FUNCTION "FC13 - MANUAL" : VOID	// FC 13
TITLE = Manual commands
VERSION : 0.1
BEGIN
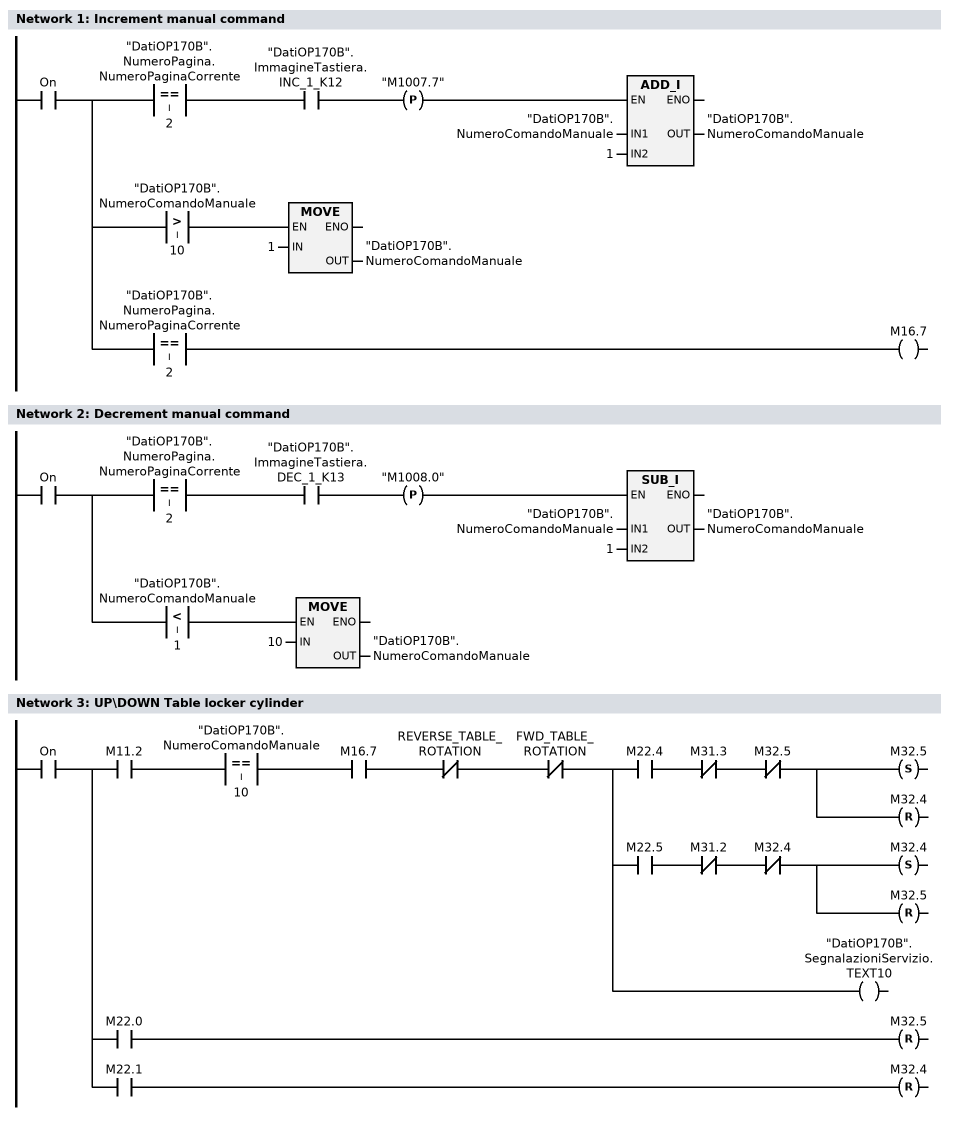
NETWORK
TITLE = Increment manual command
      A     "On";
      =     L 1.0;
      A     L 1.0;
      A(;
      L     "DatiOP170B".NumeroPagina.NumeroPaginaCorrente;
      L     2;
      ==I;
      );
      A     "DatiOP170B".ImmagineTastiera.INC_1_K12;
      FP    "M1007.7";
      JNB   _001;
      L     "DatiOP170B".NumeroComandoManuale;
      L     1;
      +I;
      T     "DatiOP170B".NumeroComandoManuale;
_001: NOP   0;
      A     L 1.0;
      A(;
      L     "DatiOP170B".NumeroComandoManuale;
      L     10;
      >I;
      );
      JNB   _002;
      L     1;
      T     "DatiOP170B".NumeroComandoManuale;
_002: NOP   0;
      A     L 1.0;
      A(;
      L     "DatiOP170B".NumeroPagina.NumeroPaginaCorrente;
      L     2;
      ==I;
      );
      =     "M16.7";
NETWORK
TITLE = Decrement manual command
      A     "On";
      =     L 1.0;
      A     L 1.0;
      A(;
      L     "DatiOP170B".NumeroPagina.NumeroPaginaCorrente;
      L     2;
      ==I;
      );
      A     "DatiOP170B".ImmagineTastiera.DEC_1_K13;
      FP    "M1008.0";
      JNB   _003;
      L     "DatiOP170B".NumeroComandoManuale;
      L     1;
      -I;
      T     "DatiOP170B".NumeroComandoManuale;
_003: NOP   0;
      A     L 1.0;
      A(;
      L     "DatiOP170B".NumeroComandoManuale;
      L     1;
      <I;
      );
      JNB   _004;
      L     10;
      T     "DatiOP170B".NumeroComandoManuale;
_004: NOP   0;
NETWORK
TITLE = UP\DOWN Table locker cylinder
      A     "On";
      =     L 1.0;
      A     L 1.0;
      A     "M11.2";
      A(;
      L     "DatiOP170B".NumeroComandoManuale;
      L     10;
      ==I;
      );
      A     "M16.7";
      AN    "REVERSE_TABLE_ROTATION";
      AN    "FWD_TABLE_ROTATION";
      =     L 1.1;
      A     L 1.1;
      A     "M22.4";
      AN    "M31.3";
      AN    "M32.5";
      S     "M32.5";
      R     "M32.4";
      A     L 1.1;
      A     "M22.5";
      AN    "M31.2";
      AN    "M32.4";
      S     "M32.4";
      R     "M32.5";
      A     L 1.1;
      BLD   102;
      =     "DatiOP170B".SegnalazioniServizio.TEXT10;
      A     L 1.0;
      A     "M22.0";
      R     "M32.5";
      A     L 1.0;
      A     "M22.1";
      R     "M32.4";
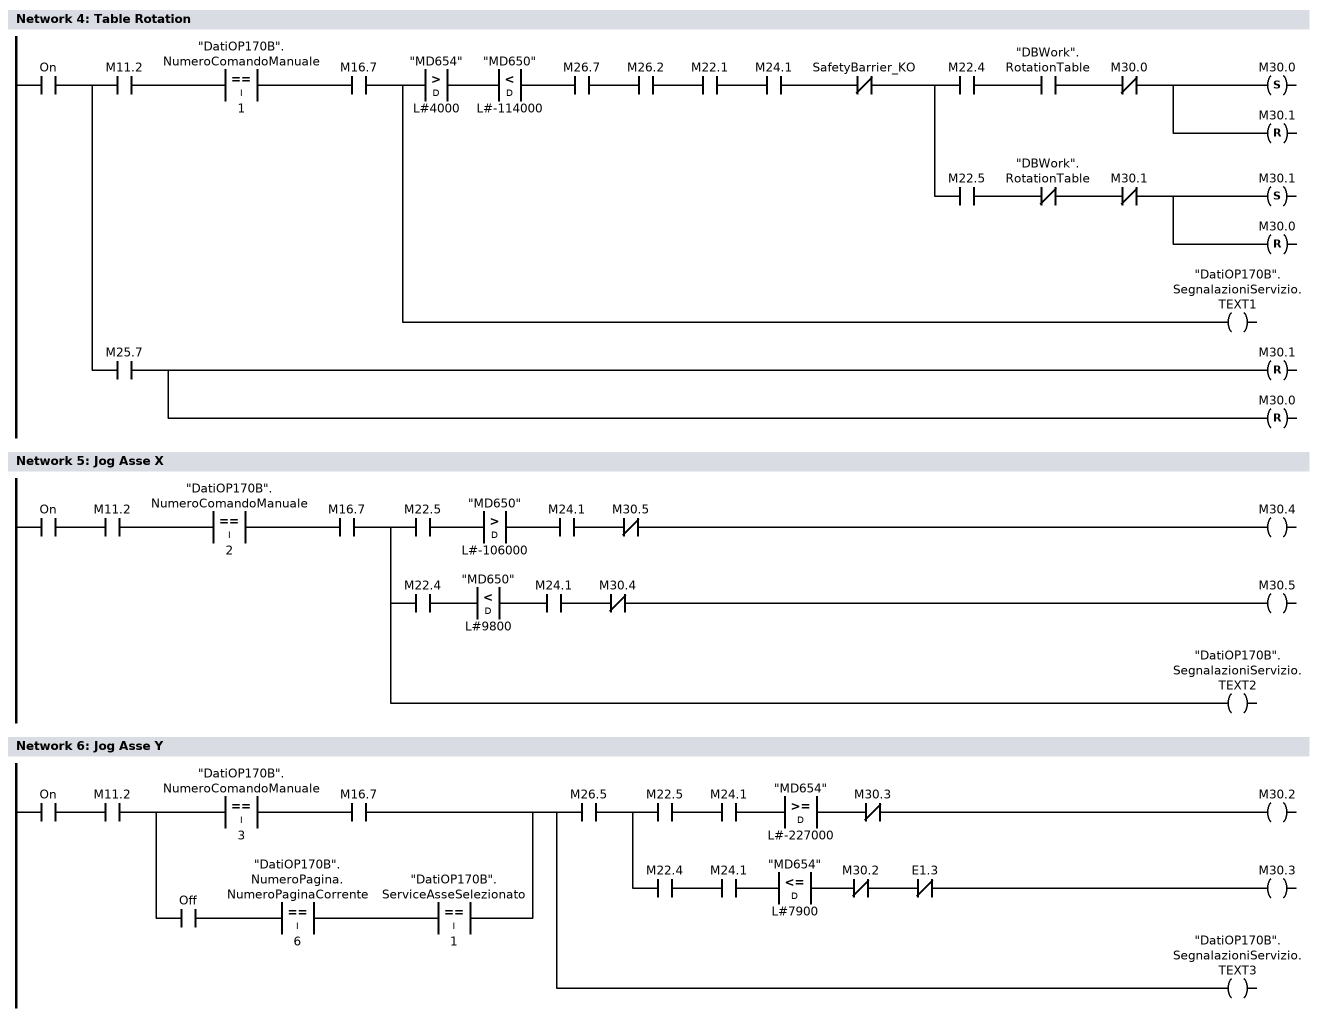
NETWORK
TITLE = Table Rotation
      A     "On";
      =     L 1.0;
      A     L 1.0;
      A     "M11.2";
      A(;
      L     "DatiOP170B".NumeroComandoManuale;
      L     1;
      ==I;
      );
      A     "M16.7";
      =     L 1.1;
      A     L 1.1;
      A(;
      L     "MD654";
      L     L#4000;
      >D;
      );
      A(;
      L     "MD650";
      L     L#-114000;
      <D;
      );
      A     "M26.7";
      A     "M26.2";
      A     "M22.1";
      A     "M24.1";
      AN    "SafetyBarrier_KO";
      =     L 1.2;
      A     L 1.2;
      A     "M22.4";
      A     "DBWork".RotationTable;
      AN    "M30.0";
      S     "M30.0";
      R     "M30.1";
      A     L 1.2;
      A     "M22.5";
      AN    "DBWork".RotationTable;
      AN    "M30.1";
      S     "M30.1";
      R     "M30.0";
      A     L 1.1;
      BLD   102;
      =     "DatiOP170B".SegnalazioniServizio.TEXT1;
      A     L 1.0;
      A     "M25.7";
      R     "M30.1";
      R     "M30.0";
NETWORK
TITLE = Jog Asse X
      A     "On";
      A     "M11.2";
      A(;
      A(;
      L     "DatiOP170B".NumeroComandoManuale;
      L     2;
      ==I;
      );
      A     "M16.7";
      );
      =     L 0.0;
      A     L 0.0;
      A     "M22.5";
      A(;
      L     "MD650";
      L     L#-106000;
      >D;
      );
      A     "M24.1";
      AN    "M30.5";
      =     "M30.4";
      A     L 0.0;
      A     "M22.4";
      A(;
      L     "MD650";
      L     L#9800;
      <D;
      );
      A     "M24.1";
      AN    "M30.4";
      =     "M30.5";
      A     L 0.0;
      BLD   102;
      =     "DatiOP170B".SegnalazioniServizio.TEXT2;
NETWORK
TITLE = Jog Asse Y
      A     "On";
      A     "M11.2";
      A(;
      A(;
      L     "DatiOP170B".NumeroComandoManuale;
      L     3;
      ==I;
      );
      A     "M16.7";
      O;
      A     "Off";
      A(;
      L     "DatiOP170B".NumeroPagina.NumeroPaginaCorrente;
      L     6;
      ==I;
      );
      A(;
      L     "DatiOP170B".ServiceAsseSelezionato;
      L     1;
      ==I;
      );
      );
      =     L 0.0;
      A     L 0.0;
      A     "M26.5";
      =     L 0.1;
      A     L 0.1;
      A     "M22.5";
      A     "M24.1";
      A(;
      L     "MD654";
      L     L#-227000;
      >=D;
      );
      AN    "M30.3";
      =     "M30.2";
      A     L 0.1;
      A     "M22.4";
      A     "M24.1";
      A(;
      L     "MD654";
      L     L#7900;
      <=D;
      );
      AN    "M30.2";
      AN    "E1.3";
      =     "M30.3";
      A     L 0.0;
      BLD   102;
      =     "DatiOP170B".SegnalazioniServizio.TEXT3;
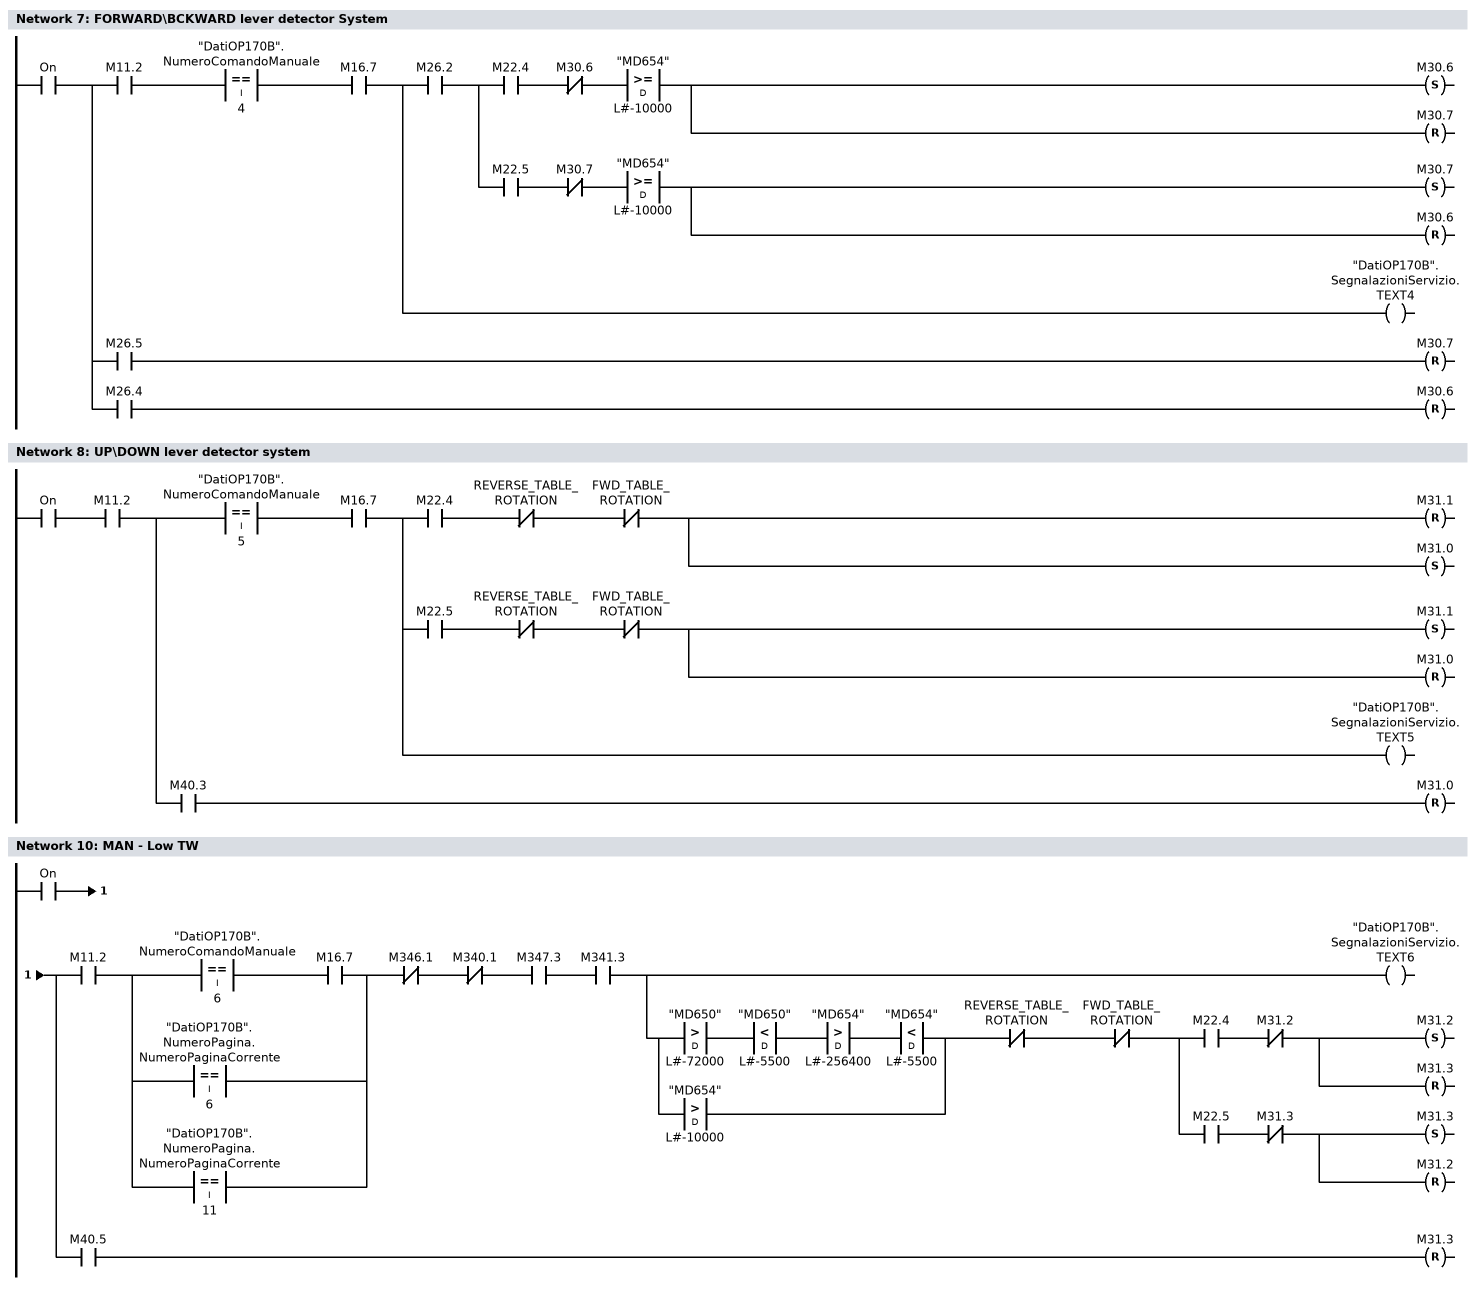
NETWORK
TITLE = FORWARD\BCKWARD lever detector System
//controllo fuori ingombro asse Y
      A     "On";
      =     L 1.0;
      A     L 1.0;
      A     "M11.2";
      A(;
      L     "DatiOP170B".NumeroComandoManuale;
      L     4;
      ==I;
      );
      A     "M16.7";
      =     L 1.1;
      A     L 1.1;
      A     "M26.2";
      =     L 1.2;
      A     L 1.2;
      A     "M22.4";
      AN    "M30.6";
      A(;
      L     "MD654";
      L     L#-10000;
      >=D;
      );
      S     "M30.6";
      R     "M30.7";
      A     L 1.2;
      A     "M22.5";
      AN    "M30.7";
      A(;
      L     "MD654";
      L     L#-10000;
      >=D;
      );
      S     "M30.7";
      R     "M30.6";
      A     L 1.1;
      BLD   102;
      =     "DatiOP170B".SegnalazioniServizio.TEXT4;
      A     L 1.0;
      A     "M26.5";
      R     "M30.7";
      A     L 1.0;
      A     "M26.4";
      R     "M30.6";
NETWORK
TITLE = UP\DOWN lever detector system
      A     "On";
      A     "M11.2";
      =     L 1.0;
      A     L 1.0;
      A(;
      L     "DatiOP170B".NumeroComandoManuale;
      L     5;
      ==I;
      );
      A     "M16.7";
      =     L 1.1;
      A     L 1.1;
      A     "M22.4";
      AN    "REVERSE_TABLE_ROTATION";
      AN    "FWD_TABLE_ROTATION";
      R     "M31.1";
      S     "M31.0";
      A     L 1.1;
      A     "M22.5";
      AN    "REVERSE_TABLE_ROTATION";
      AN    "FWD_TABLE_ROTATION";
      S     "M31.1";
      R     "M31.0";
      A     L 1.1;
      BLD   102;
      =     "DatiOP170B".SegnalazioniServizio.TEXT5;
      A     L 1.0;
      A     "M40.3";
      R     "M31.0";
NETWORK
TITLE = UP\DOWN Torch Welding Machine
//      U     "On"
//      =     L      0.0
//      U     L      0.0
//      U     "M11.2"
//      U(    
//      U(    
//      L     "DatiOP170B".NumeroComandoManuale
//      L     6
//      ==I   
//      )     
//      U     "M16.7"
//      O     
//      U(    
//      O(    
//      L     "DatiOP170B".NumeroPagina.NumeroPaginaCorrente
//      L     6
//      ==I   
//      )     
//      O(    
//      L     "DatiOP170B".NumeroPagina.NumeroPaginaCorrente
//      L     11
//      ==I   
//      )     
//      )     
//      UN    "M346.1"
//      UN    "M340.1"
//      U     "M347.3"
//      U     "M341.3"
//      )     
//      =     L      0.1
//      U     L      0.1
//      U(    
//      U(    
//      L     "MD650"
//      L     L#-72000
//      >D    
//      )     
//      U(    
//      L     "MD650"
//      L     L#-5500
//      <D    
//      )     
//      U(    
//      L     "MD654"
//      L     L#-256400
//      >D    
//      )     
//      U(    
//      L     "MD654"
//      L     L#-5500
//      <D    
//      )     
//      O(    
//      L     "MD654"
//      L     -10000
//      >D    
//      )     
//      )     
//      UN    "REVERSE_TABLE_ROTATION"
//      UN    "FWD_TABLE_ROTATION"
//      =     L      0.2
//      U     L      0.2
//      U     "M22.4"
//      UN    "M31.2"
//      S     "M31.2"
//      R     "M31.3"
//      U     L      0.2
//      U     "M22.5"
//      UN    "M31.3"
//      S     "M31.3"
//      R     "M31.2"
//      U     L      0.1
//      BLD   102
//      =     "DatiOP170B".SegnalazioniServizio.TEXT6
//      U     L      0.0
//      U     "M40.5"
//      R     "M31.3"
//  A     L      0.0
// A     "M24.1"
// R     "M31.2"
NETWORK
TITLE = MAN - Low TW
      A     "On";
      =     L 1.0;
      A     L 1.0;
      A     "M11.2";
      A(;
      A(;
      L     "DatiOP170B".NumeroComandoManuale;
      L     6;
      ==I;
      );
      A     "M16.7";
      O(;
      L     "DatiOP170B".NumeroPagina.NumeroPaginaCorrente;
      L     6;
      ==I;
      );
      O(;
      L     "DatiOP170B".NumeroPagina.NumeroPaginaCorrente;
      L     11;
      ==I;
      );
      );
      AN    "M346.1";
      AN    "M340.1";
      A     "M347.3";
      A     "M341.3";
      =     L 1.1;
      A     L 1.1;
      BLD   102;
      =     "DatiOP170B".SegnalazioniServizio.TEXT6;
      A     L 1.1;
      A(;
      A(;
      L     "MD650";
      L     L#-72000;
      >D;
      );
      A(;
      L     "MD650";
      L     L#-5500;
      <D;
      );
      A(;
      L     "MD654";
      L     L#-256400;
      >D;
      );
      A(;
      L     "MD654";
      L     L#-5500;
      <D;
      );
      O(;
      L     "MD654";
      L     L#-10000;
      >D;
      );
      );
      AN    "REVERSE_TABLE_ROTATION";
      AN    "FWD_TABLE_ROTATION";
      =     L 1.2;
      A     L 1.2;
      A     "M22.4";
      AN    "M31.2";
      S     "M31.2";
      R     "M31.3";
      A     L 1.2;
      A     "M22.5";
      AN    "M31.3";
      S     "M31.3";
      R     "M31.2";
      A     L 1.0;
      A     "M40.5";
      R     "M31.3";
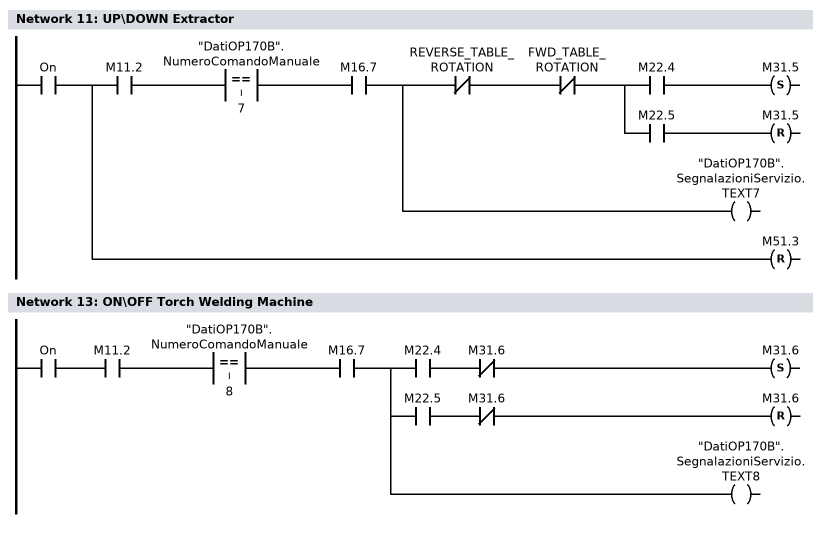
NETWORK
TITLE = UP\DOWN Extractor
      A     "On";
      =     L 1.0;
      A     L 1.0;
      A     "M11.2";
      A(;
      L     "DatiOP170B".NumeroComandoManuale;
      L     7;
      ==I;
      );
      A     "M16.7";
      =     L 1.1;
      A     L 1.1;
      AN    "REVERSE_TABLE_ROTATION";
      AN    "FWD_TABLE_ROTATION";
      =     L 1.2;
      A     L 1.2;
      A     "M22.4";
      S     "M31.5";
      A     L 1.2;
      A     "M22.5";
      R     "M31.5";
      A     L 1.1;
      BLD   102;
      =     "DatiOP170B".SegnalazioniServizio.TEXT7;
      A     L 1.0;
      BLD   102;
      R     "M51.3";
NETWORK
TITLE =
NETWORK
TITLE = ON\OFF Torch Welding Machine
      A     "On";
      A     "M11.2";
      A(;
      L     "DatiOP170B".NumeroComandoManuale;
      L     8;
      ==I;
      );
      A     "M16.7";
      =     L 1.0;
      A     L 1.0;
      A     "M22.4";
      AN    "M31.6";
      S     "M31.6";
      A     L 1.0;
      A     "M22.5";
      AN    "M31.6";
      R     "M31.6";
      A     L 1.0;
      BLD   102;
      =     "DatiOP170B".SegnalazioniServizio.TEXT8;
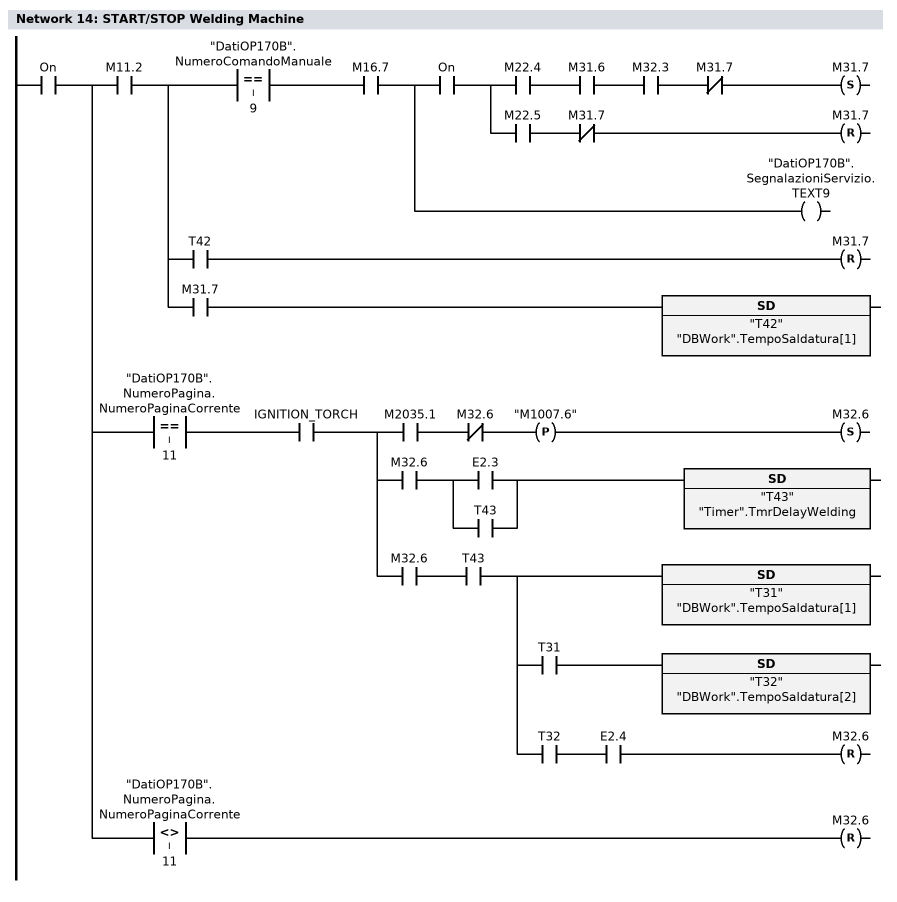
NETWORK
TITLE = START/STOP Welding Machine
      A     "On";
      =     L 1.0;
      A     L 1.0;
      A     "M11.2";
      =     L 1.1;
      A     L 1.1;
      A(;
      L     "DatiOP170B".NumeroComandoManuale;
      L     9;
      ==I;
      );
      A     "M16.7";
      =     L 1.2;
      A     L 1.2;
      A     "On";
      =     L 1.3;
      A     L 1.3;
      A     "M22.4";
      A     "M31.6";
      A     "M32.3";
      AN    "M31.7";
      S     "M31.7";
      A     L 1.3;
      A     "M22.5";
      AN    "M31.7";
      R     "M31.7";
      A     L 1.2;
      BLD   102;
      =     "DatiOP170B".SegnalazioniServizio.TEXT9;
      A     L 1.1;
      A     "T42";
      R     "M31.7";
      A     L 1.1;
      A     "M31.7";
      L     "DBWork".TempoSaldatura[1];
      SD    "T42";
      A     L 1.0;
      A(;
      L     "DatiOP170B".NumeroPagina.NumeroPaginaCorrente;
      L     11;
      ==I;
      );
      A     "IGNITION_TORCH";
      =     L 1.1;
      A     L 1.1;
      A     "M2035.1";
      AN    "M32.6";
      FP    "M1007.6";
      S     "M32.6";
      A     L 1.1;
      A     "M32.6";
      A(;
      O     "E2.3";
      O     "T43";
      );
      L     "Timer".TmrDelayWelding;
      SD    "T43";
      A     L 1.1;
      A     "M32.6";
      A     "T43";
      =     L 1.2;
      A     L 1.2;
      BLD   102;
      L     "DBWork".TempoSaldatura[1];
      SD    "T31";
      A     L 1.2;
      A     "T31";
      L     "DBWork".TempoSaldatura[2];
      SD    "T32";
      A     L 1.2;
      A     "T32";
      A     "E2.4";
      R     "M32.6";
      A     L 1.0;
      A(;
      L     "DatiOP170B".NumeroPagina.NumeroPaginaCorrente;
      L     11;
      <>I;
      );
      R     "M32.6";
END_FUNCTION

FUNCTION "FC14 - AUTOMATIC" : VOID	// FC 14
TITLE = Automatic cycle management
VERSION : 0.1
VAR_TEMP
  MinX : DINT ;
  MinY : DINT ;
  MaxX : DINT ;
  MaxY : DINT ;
END_VAR
BEGIN
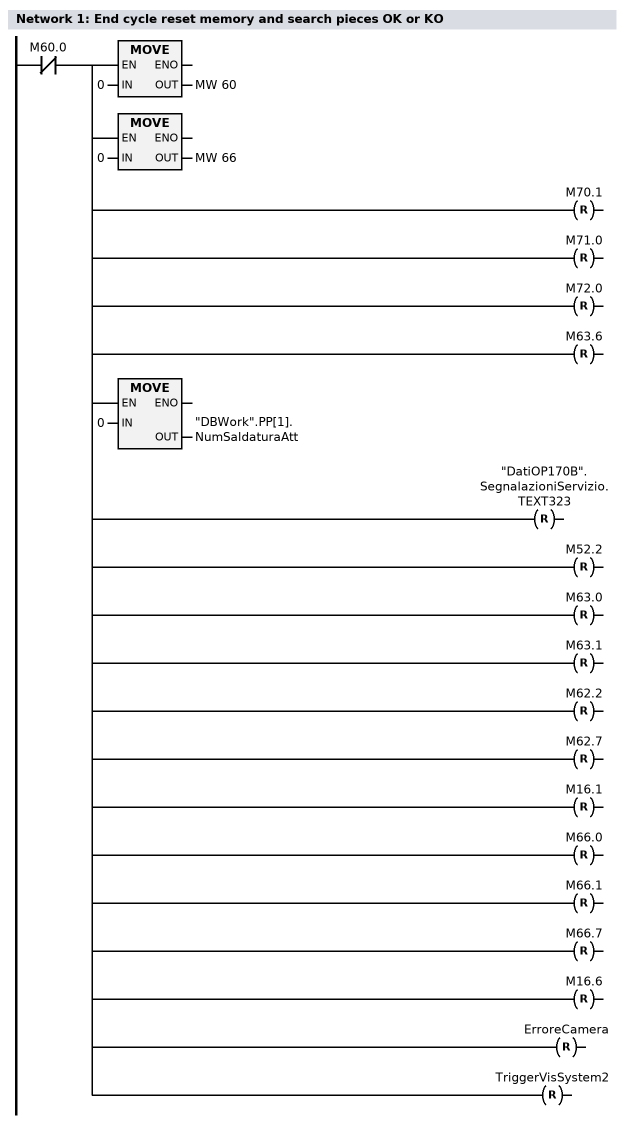
NETWORK
TITLE = End cycle reset memory and search pieces OK or KO
      AN    "M60.0";
      =     L 16.0;
      A     L 16.0;
      JNB   _001;
      L     0;
      T     MW 60;
_001: NOP   0;
      A     L 16.0;
      JNB   _002;
      L     0;
      T     MW 66;
_002: NOP   0;
      A     L 16.0;
      BLD   102;
      R     "M70.1";
      A     L 16.0;
      BLD   102;
      R     "M71.0";
      A     L 16.0;
      BLD   102;
      R     "M72.0";
      A     L 16.0;
      BLD   102;
      R     "M63.6";
      A     L 16.0;
      JNB   _003;
      L     0;
      T     "DBWork".PP[1].NumSaldaturaAtt;
_003: NOP   0;
      A     L 16.0;
      BLD   102;
      R     "DatiOP170B".SegnalazioniServizio.TEXT323;
      A     L 16.0;
      BLD   102;
      R     "M52.2";
      A     L 16.0;
      BLD   102;
      R     "M63.0";
      A     L 16.0;
      BLD   102;
      R     "M63.1";
      A     L 16.0;
      BLD   102;
      R     "M62.2";
      A     L 16.0;
      BLD   102;
      R     "M62.7";
      A     L 16.0;
      BLD   102;
      R     "M16.1";
      A     L 16.0;
      BLD   102;
      R     "M66.0";
      A     L 16.0;
      BLD   102;
      R     "M66.1";
      A     L 16.0;
      BLD   102;
      R     "M66.7";
      A     L 16.0;
      BLD   102;
      R     "M16.6";
      A     L 16.0;
      BLD   102;
      R     "ErroreCamera";
      A     L 16.0;
      BLD   102;
      R     "TriggerVisSystem2";
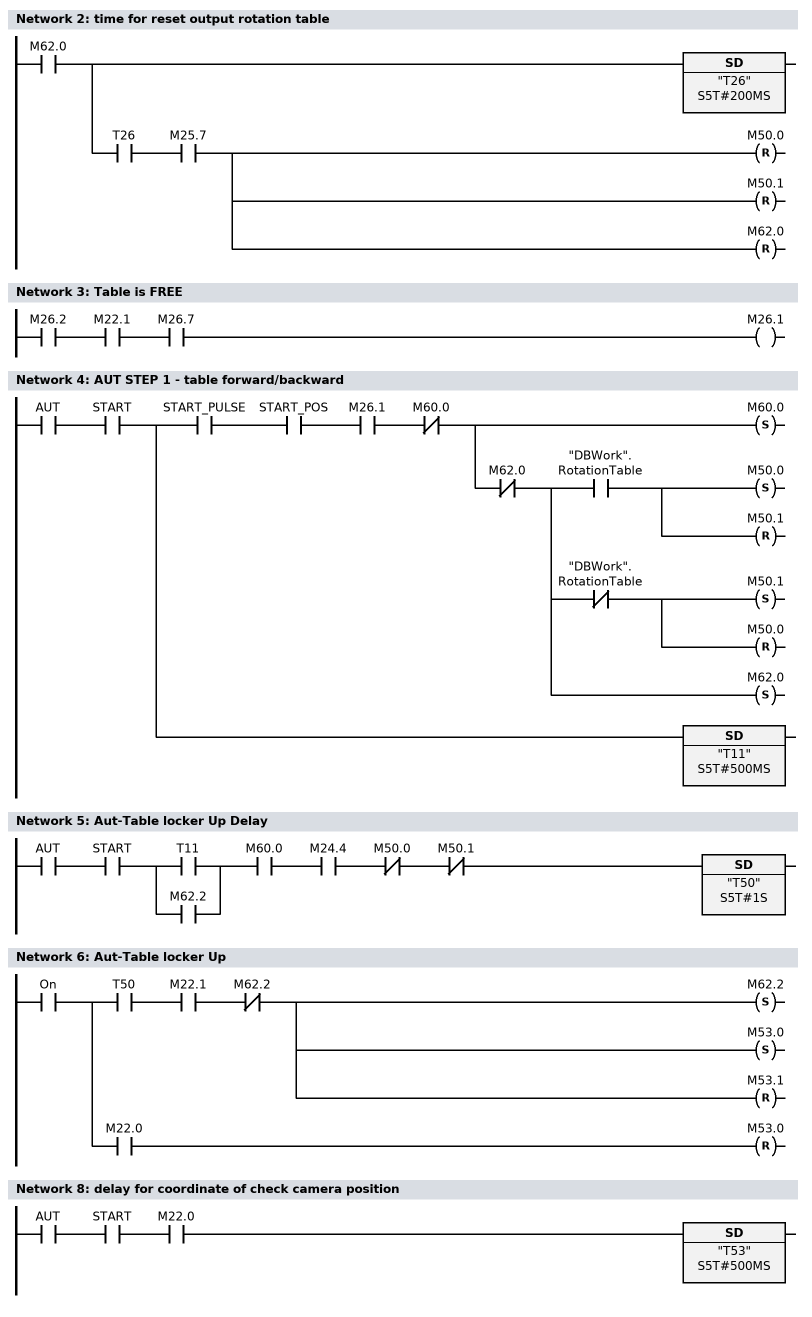
NETWORK
TITLE = time for reset output rotation table
//Reset Output Rotation Table 
      A     "M62.0";
      =     L 16.0;
      A     L 16.0;
      BLD   102;
      L     S5T#200MS;
      SD    "T26";
      A     L 16.0;
      A     "T26";
      A     "M25.7";
      R     "M50.0";
      R     "M50.1";
      R     "M62.0";
NETWORK
TITLE = Table is FREE
      A     "M26.2";
      A     "M22.1";
      A     "M26.7";
      =     "M26.1";
NETWORK
TITLE = AUT STEP 1 - table forward/backward
      A     "AUT";
      A     "START";
      =     L 16.0;
      A     L 16.0;
      A     "START_PULSE";
      A     "START_POS";
      A     "M26.1";
      AN    "M60.0";
      =     L 16.1;
      A     L 16.1;
      BLD   102;
      S     "M60.0";
      A     L 16.1;
      AN    "M62.0";
      =     L 16.2;
      A     L 16.2;
      A     "DBWork".RotationTable;
      S     "M50.0";
      R     "M50.1";
      A     L 16.2;
      AN    "DBWork".RotationTable;
      S     "M50.1";
      R     "M50.0";
      A     L 16.2;
      BLD   102;
      S     "M62.0";
      A     L 16.0;
      BLD   102;
      L     S5T#500MS;
      SD    "T11";
NETWORK
TITLE = Aut-Table locker Up Delay
      A     "AUT";
      A     "START";
      A(;
      O     "T11";
      O     "M62.2";
      );
      A     "M60.0";
      A     "M24.4";
      AN    "M50.0";
      AN    "M50.1";
      L     S5T#1S;
      SD    "T50";
NETWORK
TITLE = Aut-Table locker Up
      A     "On";
      =     L 16.0;
      A     L 16.0;
      A     "T50";
      A     "M22.1";
      AN    "M62.2";
      S     "M62.2";
      S     "M53.0";
      R     "M53.1";
      A     L 16.0;
      A     "M22.0";
      R     "M53.0";
NETWORK
TITLE = Check With OMRON if Component is OK
NETWORK
TITLE = delay for coordinate of check camera position
      A     "AUT";
      A     "START";
      A     "M22.0";
      L     S5T#500MS;
      SD    "T53";
NETWORK
TITLE =
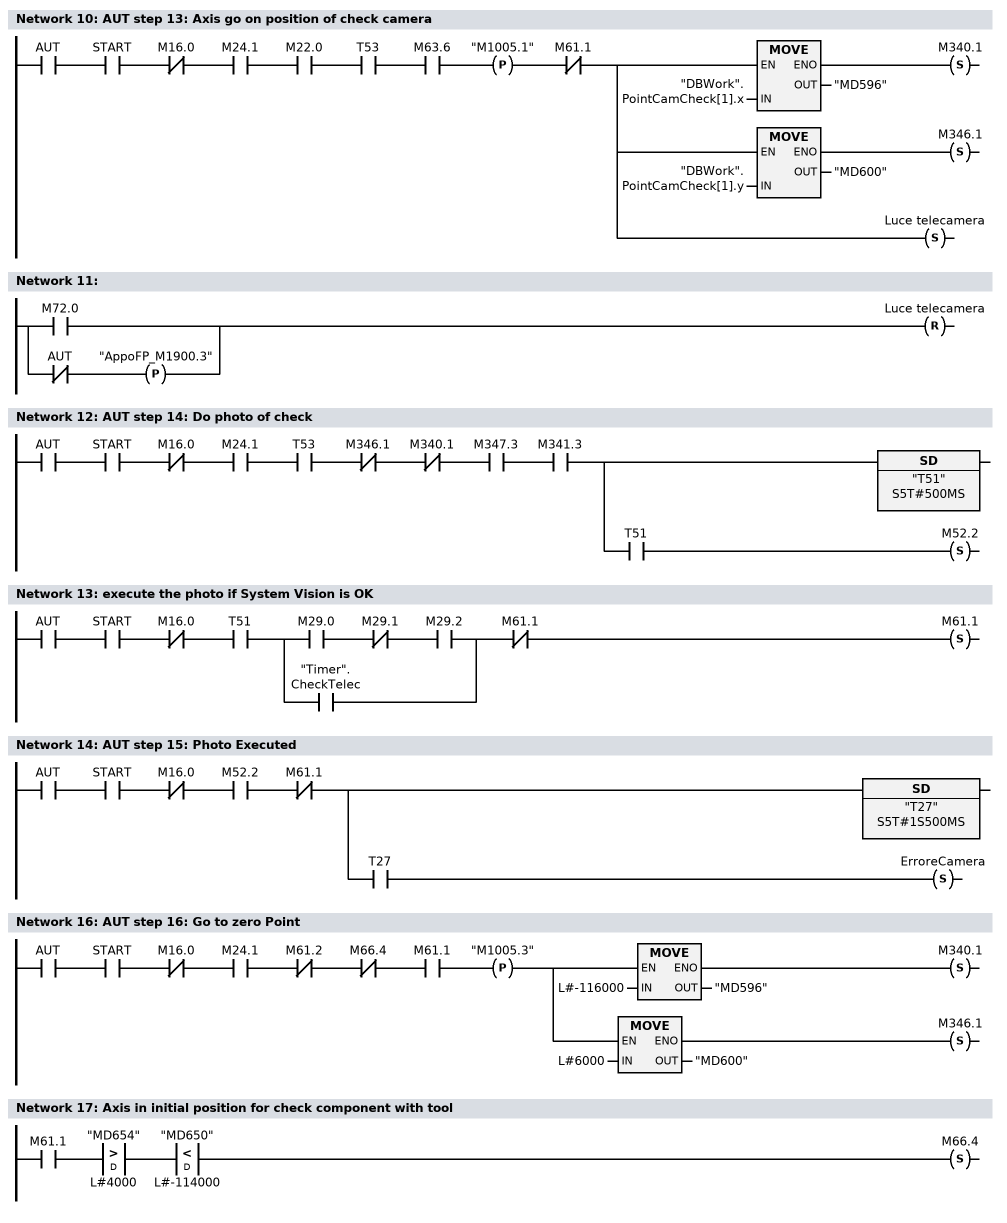
NETWORK
TITLE = AUT step 13: Axis go on position of check camera
      A     "AUT";
      A     "START";
      AN    "M16.0";
      A     "M24.1";
      A     "M22.0";
      A     "T53";
      A     "M63.6";
      FP    "M1005.1";
      AN    "M61.1";
      =     L 16.0;
      A     L 16.0;
      JNB   _004;
      L     "DBWork".PointCamCheck[1].x;
      T     "MD596";
      SET;
      SAVE;
      CLR;
_004: A     BR;
      S     "M340.1";
      A     L 16.0;
      JNB   _005;
      L     "DBWork".PointCamCheck[1].y;
      T     "MD600";
      SET;
      SAVE;
      CLR;
_005: A     BR;
      S     "M346.1";
      A     L 16.0;
      BLD   102;
      S     "Luce telecamera";
NETWORK
TITLE =
      O     "M72.0";
      O(;
      AN    "AUT";
      FP    "AppoFP_M1900.3";
      );
      R     "Luce telecamera";
NETWORK
TITLE = AUT step 14: Do photo of check 
      A     "AUT";
      A     "START";
      AN    "M16.0";
      A     "M24.1";
      A     "T53";
      AN    "M346.1";
      AN    "M340.1";
      A     "M347.3";
      A     "M341.3";
      =     L 16.0;
      A     L 16.0;
      BLD   102;
      L     S5T#500MS;
      SD    "T51";
      A     L 16.0;
      A     "T51";
      S     "M52.2";
NETWORK
TITLE = execute the photo if System Vision is OK
      A     "AUT";
      A     "START";
      AN    "M16.0";
      A     "T51";
      A(;
      A     "M29.0";
      AN    "M29.1";
      A     "M29.2";
      O     "Timer".CheckTelec;
      );
      AN    "M61.1";
      S     "M61.1";
NETWORK
TITLE = AUT step 15: Photo Executed
      A     "AUT";
      A     "START";
      AN    "M16.0";
      A     "M52.2";
      AN    "M61.1";
      =     L 16.0;
      A     L 16.0;
      BLD   102;
      L     S5T#1S500MS;
      SD    "T27";
      A     L 16.0;
      A     "T27";
      S     "ErroreCamera";
NETWORK
TITLE =
NETWORK
TITLE = AUT step 16: Go to zero Point
      A     "AUT";
      A     "START";
      AN    "M16.0";
      A     "M24.1";
      AN    "M61.2";
      AN    "M66.4";
      A     "M61.1";
      FP    "M1005.3";
      =     L 16.0;
      A     L 16.0;
      JNB   _006;
      L     L#-116000;
      T     "MD596";
      SET;
      SAVE;
      CLR;
_006: A     BR;
      S     "M340.1";
      A     L 16.0;
      JNB   _007;
      L     L#6000;
      T     "MD600";
      SET;
      SAVE;
      CLR;
_007: A     BR;
      S     "M346.1";
NETWORK
TITLE = Axis in initial position for check component with tool
      A     "M61.1";
      A(;
      L     "MD654";
      L     L#4000;
      >D;
      );
      A(;
      L     "MD650";
      L     L#-114000;
      <D;
      );
      S     "M66.4";
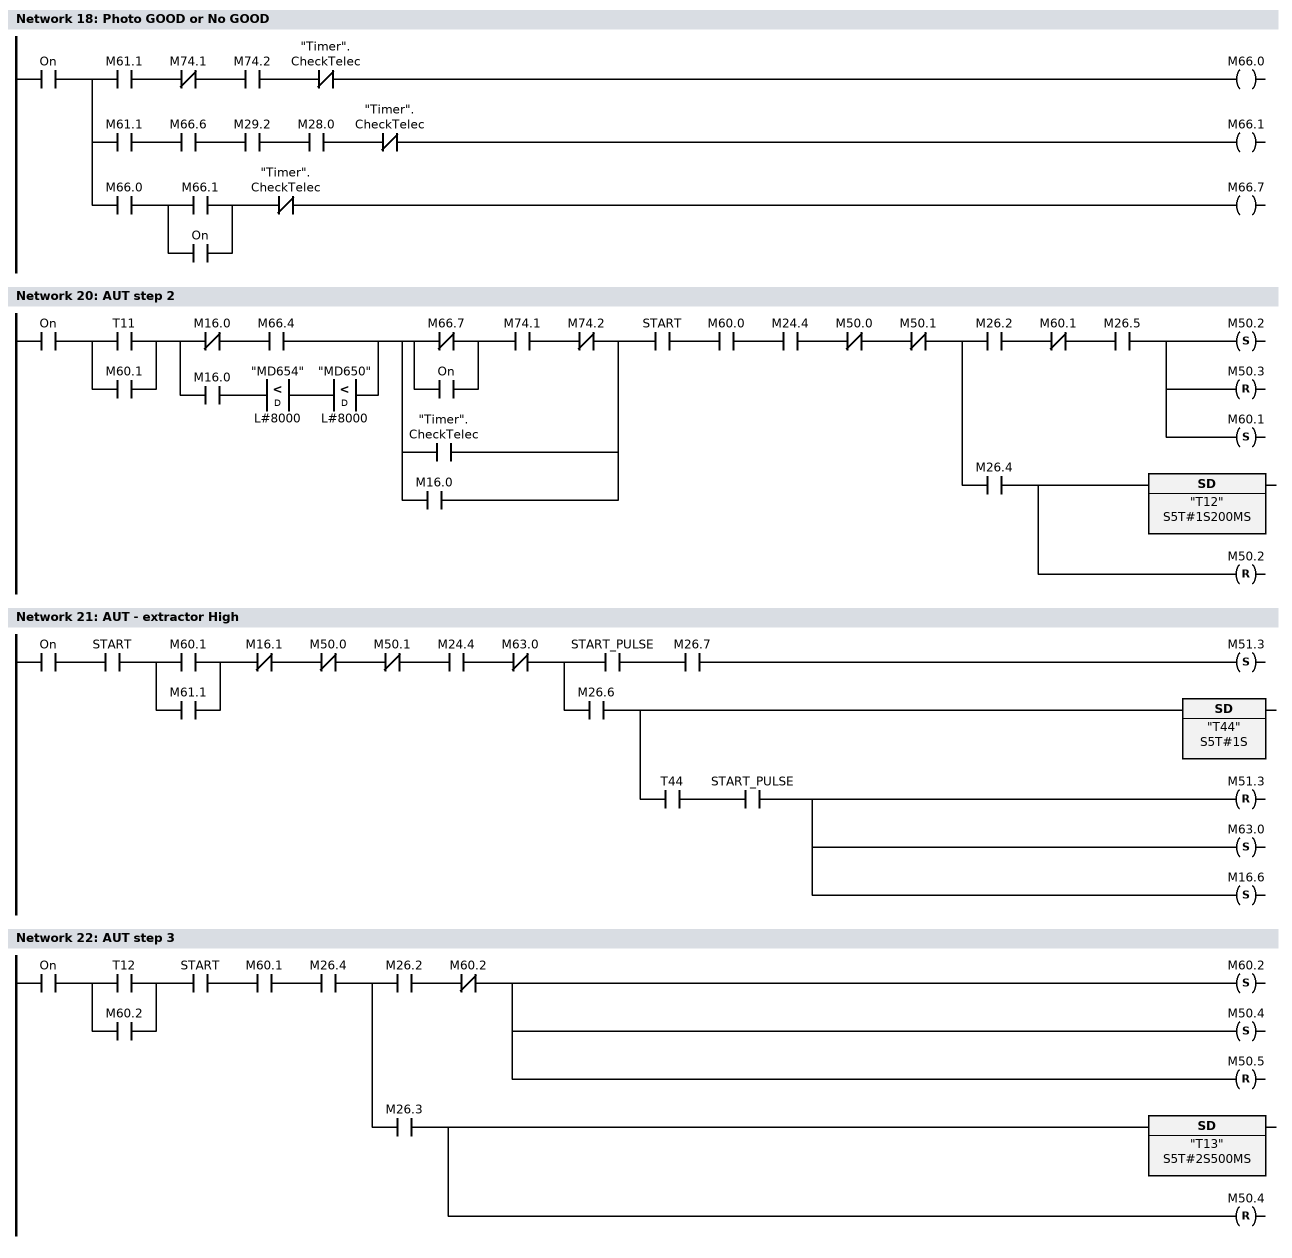
NETWORK
TITLE = Photo GOOD or No GOOD
      A     "On";
      =     L 16.0;
      A     L 16.0;
      A     "M61.1";
      AN    "M74.1";
      A     "M74.2";
      AN    "Timer".CheckTelec;
      =     "M66.0";
      A     L 16.0;
      A     "M61.1";
      A     "M66.6";
      A     "M29.2";
      A     "M28.0";
      AN    "Timer".CheckTelec;
      =     "M66.1";
      A     L 16.0;
      A     "M66.0";
      A(;
      O     "M66.1";
      O     "On";
      );
      AN    "Timer".CheckTelec;
      =     "M66.7";
NETWORK
TITLE =
NETWORK
TITLE = AUT step 2
//Step 2: System Detector Forward ed 
      A     "On";
      A(;
      O     "T11";
      O     "M60.1";
      );
      A(;
      AN    "M16.0";
      A     "M66.4";
      O;
      A     "M16.0";
      A(;
      L     "MD654";
      L     L#8000;
      <D;
      );
      A(;
      L     "MD650";
      L     L#8000;
      <D;
      );
      );
      A(;
      A(;
      ON    "M66.7";
      O     "On";
      );
      A     "M74.1";
      AN    "M74.2";
      O     "Timer".CheckTelec;
      O     "M16.0";
      );
      A     "START";
      A     "M60.0";
      A     "M24.4";
      AN    "M50.0";
      AN    "M50.1";
      =     L 16.0;
      A     L 16.0;
      A     "M26.2";
      AN    "M60.1";
      A     "M26.5";
      S     "M50.2";
      R     "M50.3";
      S     "M60.1";
      A     L 16.0;
      A     "M26.4";
      L     S5T#1S200MS;
      SD    "T12";
      R     "M50.2";
NETWORK
TITLE = AUT - extractor High
//Insert Extractor , extract worked pieces, i make it together Step 2
      A     "On";
      A     "START";
      A(;
      O     "M60.1";
      O     "M61.1";
      );
      AN    "M16.1";
      AN    "M50.0";
      AN    "M50.1";
      A     "M24.4";
      AN    "M63.0";
      =     L 16.0;
      A     L 16.0;
      A     "START_PULSE";
      A     "M26.7";
      S     "M51.3";
      A     L 16.0;
      A     "M26.6";
      =     L 16.1;
      A     L 16.1;
      BLD   102;
      L     S5T#1S;
      SD    "T44";
      A     L 16.1;
      A     "T44";
      A     "START_PULSE";
      R     "M51.3";
      S     "M63.0";
      S     "M16.6";
NETWORK
TITLE = AUT step 3
//Step 3: System Detector Low
      A     "On";
      A(;
      O     "T12";
      O     "M60.2";
      );
      A     "START";
      A     "M60.1";
      A     "M26.4";
      =     L 16.0;
      A     L 16.0;
      A     "M26.2";
      AN    "M60.2";
      S     "M60.2";
      S     "M50.4";
      R     "M50.5";
      A     L 16.0;
      A     "M26.3";
      L     S5T#2S500MS;
      SD    "T13";
      R     "M50.4";
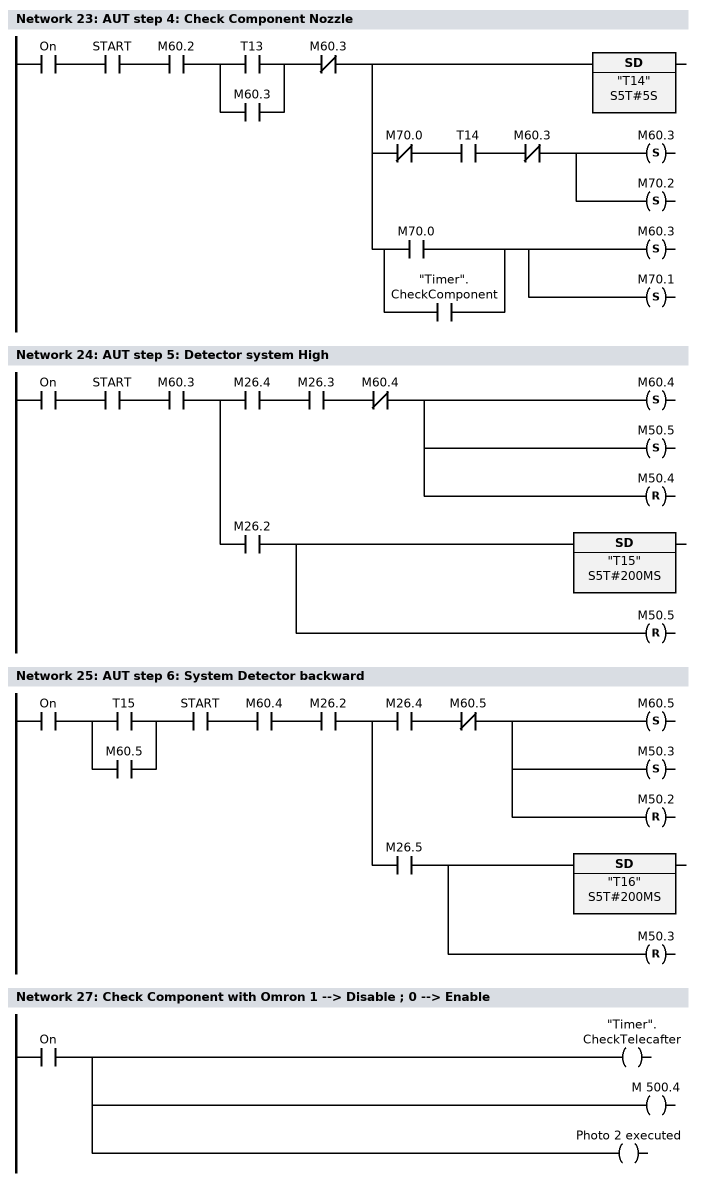
NETWORK
TITLE = AUT step 4: Check Component Nozzle
//check if is possible work pieces
//
      A     "On";
      A     "START";
      A     "M60.2";
      A(;
      O     "T13";
      O     "M60.3";
      );
      AN    "M60.3";
      =     L 16.0;
      A     L 16.0;
      BLD   102;
      L     S5T#5S;
      SD    "T14";
      A     L 16.0;
      AN    "M70.0";
      A     "T14";
      AN    "M60.3";
      S     "M60.3";
      S     "M70.2";
      A     L 16.0;
      A(;
      O     "M70.0";
      O     "Timer".CheckComponent;
      );
      S     "M60.3";
      S     "M70.1";
NETWORK
TITLE = AUT step 5: Detector system High
      A     "On";
      A     "START";
      A     "M60.3";
      =     L 16.0;
      A     L 16.0;
      A     "M26.4";
      A     "M26.3";
      AN    "M60.4";
      S     "M60.4";
      S     "M50.5";
      R     "M50.4";
      A     L 16.0;
      A     "M26.2";
      L     S5T#200MS;
      SD    "T15";
      R     "M50.5";
NETWORK
TITLE = AUT step 6: System Detector backward
//torno con il controllo in posizione iniziale
      A     "On";
      A(;
      O     "T15";
      O     "M60.5";
      );
      A     "START";
      A     "M60.4";
      A     "M26.2";
      =     L 16.0;
      A     L 16.0;
      A     "M26.4";
      AN    "M60.5";
      S     "M60.5";
      S     "M50.3";
      R     "M50.2";
      A     L 16.0;
      A     "M26.5";
      L     S5T#200MS;
      SD    "T16";
      R     "M50.3";
NETWORK
TITLE =
NETWORK
TITLE = Check Component with Omron 1 --> Disable ; 0 --> Enable
      A     "On";
      =     "Timer".CheckTelecafter;
      =     M 500.4;
      =     "Photo 2 executed";
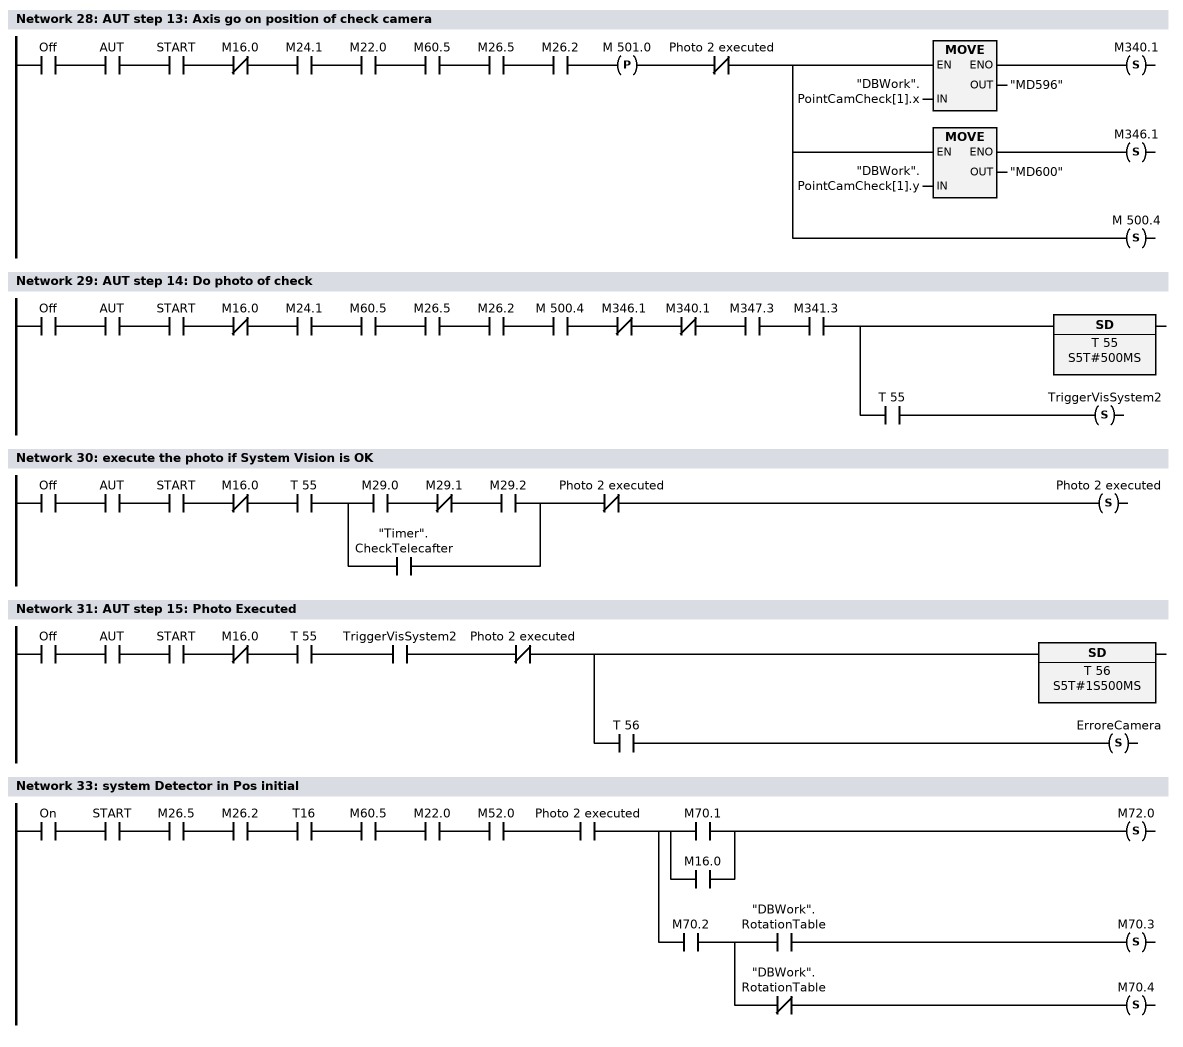
NETWORK
TITLE = AUT step 13: Axis go on position of check camera
      A     "Off";
      A     "AUT";
      A     "START";
      AN    "M16.0";
      A     "M24.1";
      A     "M22.0";
      A     "M60.5";
      A     "M26.5";
      A     "M26.2";
      FP    M 501.0;
      AN    "Photo 2 executed";
      =     L 16.0;
      A     L 16.0;
      JNB   _008;
      L     "DBWork".PointCamCheck[1].x;
      T     "MD596";
      SET;
      SAVE;
      CLR;
_008: A     BR;
      S     "M340.1";
      A     L 16.0;
      JNB   _009;
      L     "DBWork".PointCamCheck[1].y;
      T     "MD600";
      SET;
      SAVE;
      CLR;
_009: A     BR;
      S     "M346.1";
      A     L 16.0;
      BLD   102;
      S     M 500.4;
NETWORK
TITLE = AUT step 14: Do photo of check 
      A     "Off";
      A     "AUT";
      A     "START";
      AN    "M16.0";
      A     "M24.1";
      A     "M60.5";
      A     "M26.5";
      A     "M26.2";
      A     M 500.4;
      AN    "M346.1";
      AN    "M340.1";
      A     "M347.3";
      A     "M341.3";
      =     L 16.0;
      A     L 16.0;
      BLD   102;
      L     S5T#500MS;
      SD    T 55;
      A     L 16.0;
      A     T 55;
      S     "TriggerVisSystem2";
NETWORK
TITLE = execute the photo if System Vision is OK
      A     "Off";
      A     "AUT";
      A     "START";
      AN    "M16.0";
      A     T 55;
      A(;
      A     "M29.0";
      AN    "M29.1";
      A     "M29.2";
      O     "Timer".CheckTelecafter;
      );
      AN    "Photo 2 executed";
      S     "Photo 2 executed";
NETWORK
TITLE = AUT step 15: Photo Executed
      A     "Off";
      A     "AUT";
      A     "START";
      AN    "M16.0";
      A     T 55;
      A     "TriggerVisSystem2";
      AN    "Photo 2 executed";
      =     L 16.0;
      A     L 16.0;
      BLD   102;
      L     S5T#1S500MS;
      SD    T 56;
      A     L 16.0;
      A     T 56;
      S     "ErroreCamera";
NETWORK
TITLE =
NETWORK
TITLE = system Detector in Pos initial
//System Detector in Pos initial and ready for detect Welding point
      A     "On";
      A     "START";
      A     "M26.5";
      A     "M26.2";
      A     "T16";
      A     "M60.5";
      A     "M22.0";
      A     "M52.0";
      A     "Photo 2 executed";
      =     L 16.0;
      A     L 16.0;
      A(;
      O     "M70.1";
      O     "M16.0";
      );
      S     "M72.0";
      A     L 16.0;
      A     "M70.2";
      =     L 16.1;
      A     L 16.1;
      A     "DBWork".RotationTable;
      S     "M70.3";
      A     L 16.1;
      AN    "DBWork".RotationTable;
      S     "M70.4";
NETWORK
TITLE = ------------START WITH WELDING
NETWORK
TITLE = AUT step 7: Axis on point of Welding
//AXIS X 
//AXIS Y 
//
//MD588 = SUPPORT FOR POINT X
//MD592 = SUPPORT FOR POINT Y
      A(;
      A     "AUT";
      A(;
      L     "DBWork".PP[1].NumSaldaturaAtt;
      L     0;
      ==I;
      );
      A     "M72.0";
      FP    "M1000.5";
      AN    "M60.6";
      O(;
      A     "AUT";
      A     "M61.3";
      FP    "M1000.4";
      );
      );
      A     "On";
      =     L 16.0;
      A     L 16.0;
      A     "DBWork".RotationTable;
      =     L 16.1;
      A(;
      A     L 16.1;
      JNB   _00a;
      L     "MD588";
      L     "Timer".OffsetX1;
      +D;
      T     "MD588";
      AN    OV;
      SAVE;
      CLR;
_00a: A     BR;
      );
      JNB   _00b;
      L     "MD588";
      T     "MD596";
      SET;
      SAVE;
      CLR;
_00b: A     BR;
      S     "M340.1";
      A(;
      A     L 16.1;
      JNB   _00c;
      L     "MD592";
      L     "Timer".OffsetY1;
      +D;
      T     "MD592";
      AN    OV;
      SAVE;
      CLR;
_00c: A     BR;
      );
      JNB   _00d;
      L     "MD592";
      T     "MD600";
      SET;
      SAVE;
      CLR;
_00d: A     BR;
      S     "M346.1";
      A     L 16.0;
      AN    "DBWork".RotationTable;
      =     L 16.1;
      A(;
      A     L 16.1;
      JNB   _016;
      L     "MD588";
      L     "DBWork2".OffsetX_2;
      +D;
      T     "MD588";
      AN    OV;
      SAVE;
      CLR;
_016: A     BR;
      );
      JNB   _017;
      L     "MD588";
      T     "MD596";
      SET;
      SAVE;
      CLR;
_017: A     BR;
      S     "M340.1";
      A(;
      A     L 16.1;
      JNB   _018;
      L     "MD592";
      L     "DBWork2".OffsetY_2;
      +D;
      T     "MD592";
      AN    OV;
      SAVE;
      CLR;
_018: A     BR;
      );
      JNB   _019;
      L     "MD592";
      T     "MD600";
      SET;
      SAVE;
      CLR;
_019: A     BR;
      S     "M346.1";
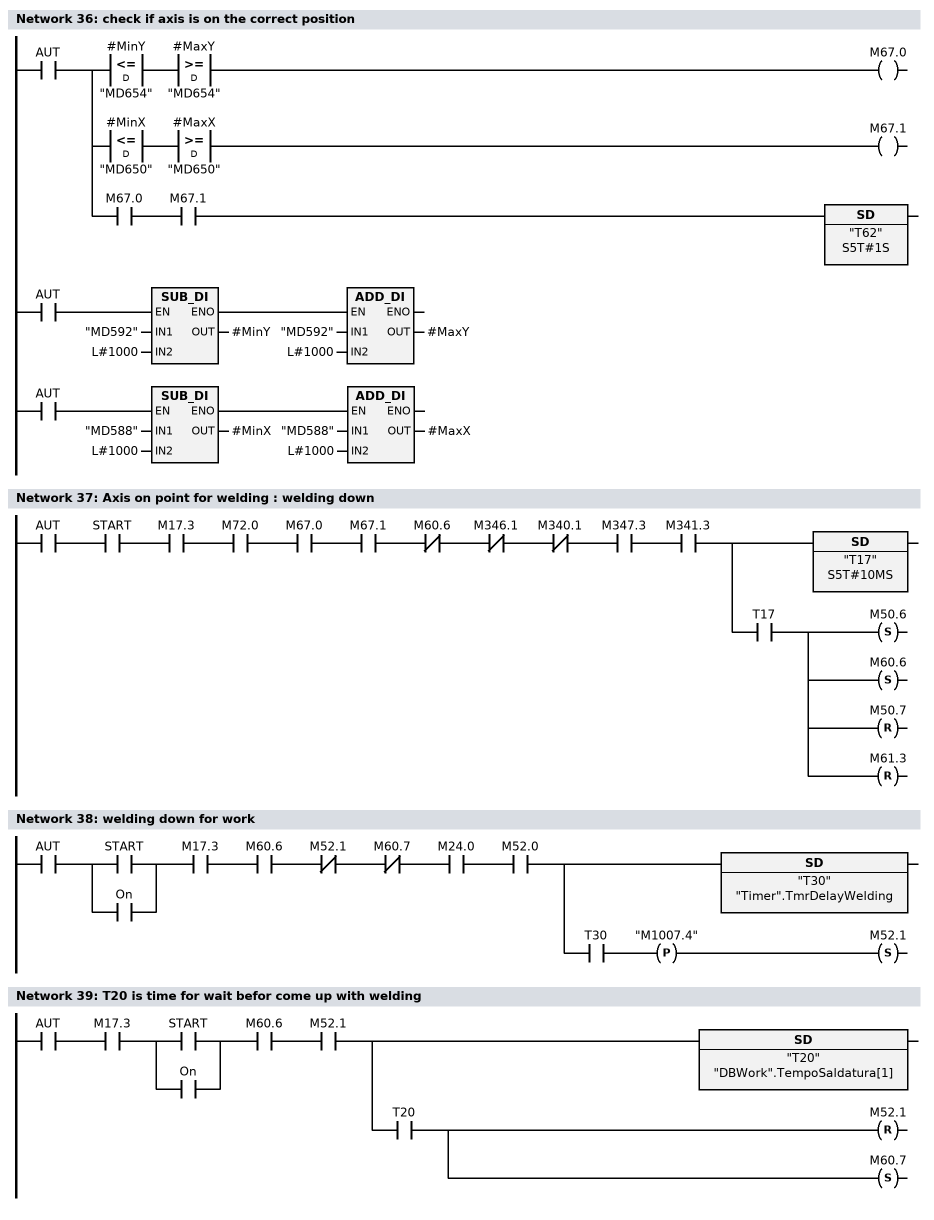
NETWORK
TITLE = check if axis is on the correct position
      A     "AUT";
      =     L 16.0;
      A(;
      A     L 16.0;
      JNB   _01a;
      L     "MD592";
      L     L#1000;
      -D;
      T     #MinY;
      AN    OV;
      SAVE;
      CLR;
_01a: A     BR;
      );
      JNB   _01b;
      L     "MD592";
      L     L#1000;
      +D;
      T     #MaxY;
_01b: NOP   0;
      A(;
      A     L 16.0;
      JNB   _01c;
      L     "MD588";
      L     L#1000;
      -D;
      T     #MinX;
      AN    OV;
      SAVE;
      CLR;
_01c: A     BR;
      );
      JNB   _01d;
      L     "MD588";
      L     L#1000;
      +D;
      T     #MaxX;
_01d: NOP   0;
      A     L 16.0;
      A(;
      L     #MinY;
      L     "MD654";
      <=D;
      );
      A(;
      L     #MaxY;
      L     "MD654";
      >=D;
      );
      =     "M67.0";
      A     L 16.0;
      A(;
      L     #MinX;
      L     "MD650";
      <=D;
      );
      A(;
      L     #MaxX;
      L     "MD650";
      >=D;
      );
      =     "M67.1";
      A     L 16.0;
      A     "M67.0";
      A     "M67.1";
      L     S5T#1S;
      SD    "T62";
NETWORK
TITLE = Axis on point for welding : welding down
//Saldatore giù
      A     "AUT";
      A     "START";
      A     "M17.3";
      A     "M72.0";
      A     "M67.0";
      A     "M67.1";
      AN    "M60.6";
      AN    "M346.1";
      AN    "M340.1";
      A     "M347.3";
      A     "M341.3";
      =     L 16.0;
      A     L 16.0;
      BLD   102;
      L     S5T#10MS;
      SD    "T17";
      A     L 16.0;
      A     "T17";
      S     "M50.6";
      S     "M60.6";
      R     "M50.7";
      R     "M61.3";
NETWORK
TITLE = welding down for work
//saldatore giu per saldatura
      A     "AUT";
      A(;
      O     "START";
      O     "On";
      );
      A     "M17.3";
      A     "M60.6";
      AN    "M52.1";
      AN    "M60.7";
      A     "M24.0";
      A     "M52.0";
      =     L 16.0;
      A     L 16.0;
      BLD   102;
      L     "Timer".TmrDelayWelding;
      SD    "T30";
      A     L 16.0;
      A     "T30";
      FP    "M1007.4";
      S     "M52.1";
NETWORK
TITLE = T20 is time for wait befor come up with welding
//Resto un tempo T20 sul punto saldato prima di rialzare la torcia
      A     "AUT";
      A     "M17.3";
      A(;
      O     "START";
      O     "On";
      );
      A     "M60.6";
      A     "M52.1";
      =     L 16.0;
      A     L 16.0;
      BLD   102;
      L     "DBWork".TempoSaldatura[1];
      SD    "T20";
      A     L 16.0;
      A     "T20";
      R     "M52.1";
      S     "M60.7";
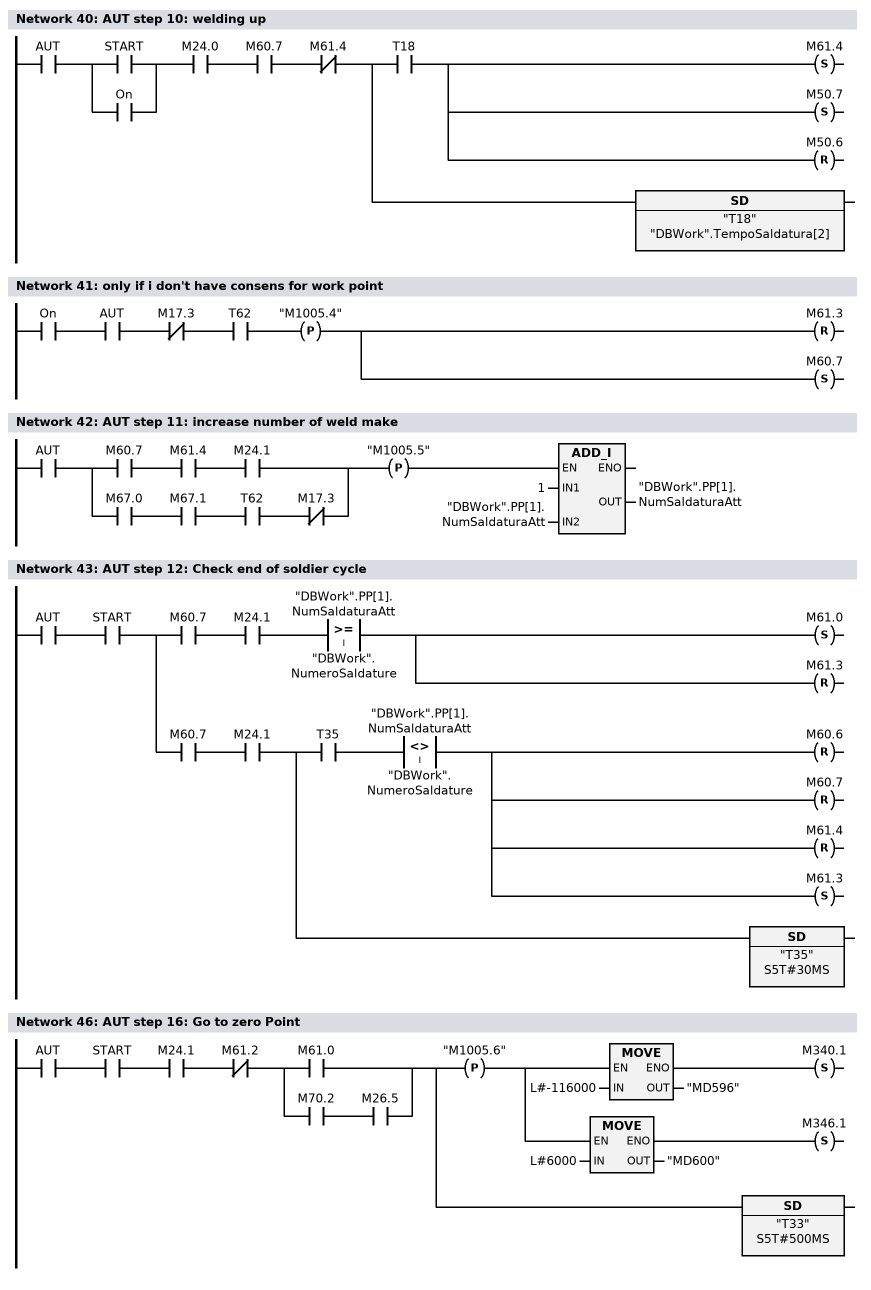
NETWORK
TITLE = AUT step 10: welding up
      A     "AUT";
      A(;
      O     "START";
      O     "On";
      );
      A     "M24.0";
      A     "M60.7";
      AN    "M61.4";
      =     L 16.0;
      A     L 16.0;
      A     "T18";
      S     "M61.4";
      S     "M50.7";
      R     "M50.6";
      A     L 16.0;
      BLD   102;
      L     "DBWork".TempoSaldatura[2];
      SD    "T18";
NETWORK
TITLE = only if i don't have consens for work point
      A     "On";
      A     "AUT";
      AN    "M17.3";
      A     "T62";
      FP    "M1005.4";
      R     "M61.3";
      S     "M60.7";
NETWORK
TITLE = AUT step 11: increase number of weld make
//incremento il numero di saldature effettuate
      A     "AUT";
      A(;
      A     "M60.7";
      A     "M61.4";
      A     "M24.1";
      O;
      A     "M67.0";
      A     "M67.1";
      A     "T62";
      AN    "M17.3";
      );
      FP    "M1005.5";
      JNB   _01e;
      L     1;
      L     "DBWork".PP[1].NumSaldaturaAtt;
      +I;
      T     "DBWork".PP[1].NumSaldaturaAtt;
_01e: NOP   0;
NETWORK
TITLE = AUT step 12: Check end of soldier cycle 
//aspetto per il passaggio delle coorddinate al simodrive
      A     "AUT";
      A     "START";
      =     L 16.0;
      A     L 16.0;
      A     "M60.7";
      A     "M24.1";
      A(;
      L     "DBWork".PP[1].NumSaldaturaAtt;
      L     "DBWork".NumeroSaldature;
      >=I;
      );
      S     "M61.0";
      R     "M61.3";
      A     L 16.0;
      A     "M60.7";
      A     "M24.1";
      =     L 16.1;
      A     L 16.1;
      A     "T35";
      A(;
      L     "DBWork".PP[1].NumSaldaturaAtt;
      L     "DBWork".NumeroSaldature;
      <>I;
      );
      R     "M60.6";
      R     "M60.7";
      R     "M61.4";
      S     "M61.3";
      A     L 16.1;
      BLD   102;
      L     S5T#30MS;
      SD    "T35";
NETWORK
TITLE =
NETWORK
TITLE =
NETWORK
TITLE = AUT step 16: Go to zero Point
      A     "AUT";
      A     "START";
      A     "M24.1";
      AN    "M61.2";
      A(;
      O     "M61.0";
      O;
      A     "M70.2";
      A     "M26.5";
      );
      =     L 16.0;
      A     L 16.0;
      FP    "M1005.6";
      =     L 16.1;
      A     L 16.1;
      JNB   _01f;
      L     L#-116000;
      T     "MD596";
      SET;
      SAVE;
      CLR;
_01f: A     BR;
      S     "M340.1";
      A     L 16.1;
      JNB   _020;
      L     L#6000;
      T     "MD600";
      SET;
      SAVE;
      CLR;
_020: A     BR;
      S     "M346.1";
      A     L 16.0;
      BLD   102;
      L     S5T#500MS;
      SD    "T33";
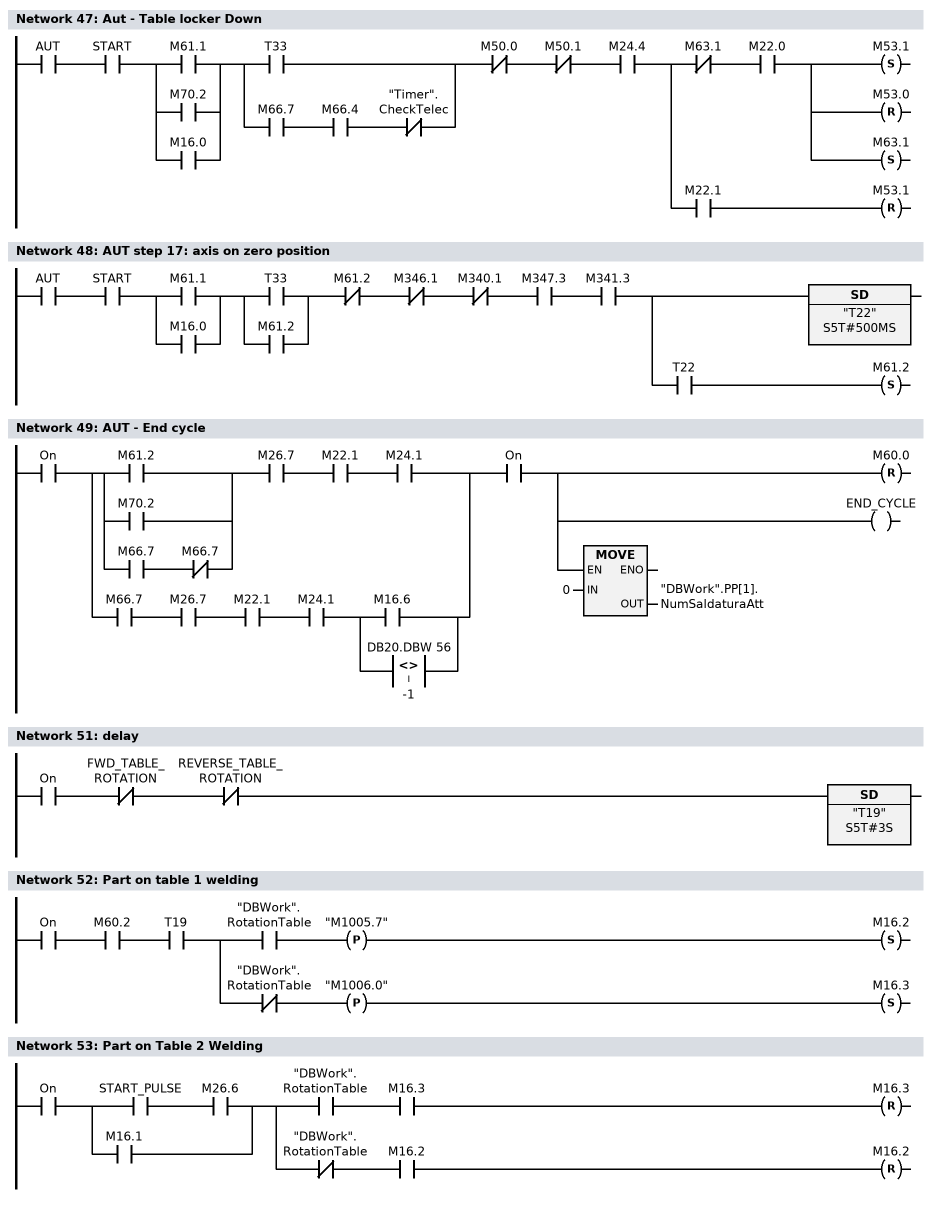
NETWORK
TITLE = Aut - Table locker Down
//Table cyclinder Low
      A     "AUT";
      A     "START";
      A(;
      O     "M61.1";
      O     "M70.2";
      O     "M16.0";
      );
      A(;
      O     "T33";
      O;
      A     "M66.7";
      A     "M66.4";
      AN    "Timer".CheckTelec;
      );
      AN    "M50.0";
      AN    "M50.1";
      A     "M24.4";
      =     L 16.0;
      A     L 16.0;
      AN    "M63.1";
      A     "M22.0";
      S     "M53.1";
      R     "M53.0";
      S     "M63.1";
      A     L 16.0;
      A     "M22.1";
      R     "M53.1";
NETWORK
TITLE = AUT step 17: axis on zero position
      A     "AUT";
      A     "START";
      A(;
      O     "M61.1";
      O     "M16.0";
      );
      A(;
      O     "T33";
      O     "M61.2";
      );
      AN    "M61.2";
      AN    "M346.1";
      AN    "M340.1";
      A     "M347.3";
      A     "M341.3";
      =     L 16.0;
      A     L 16.0;
      BLD   102;
      L     S5T#500MS;
      SD    "T22";
      A     L 16.0;
      A     "T22";
      S     "M61.2";
NETWORK
TITLE = AUT - End cycle
      A     "On";
      A(;
      A(;
      O     "M61.2";
      O     "M70.2";
      O;
      A     "M66.7";
      AN    "M66.7";
      );
      A     "M26.7";
      A     "M22.1";
      A     "M24.1";
      O;
      A     "M66.7";
      A     "M26.7";
      A     "M22.1";
      A     "M24.1";
      A(;
      O     "M16.6";
      O(;
      L     DB20.DBW 56;
      L     -1;
      <>I;
      );
      );
      );
      A     "On";
      =     L 16.0;
      A     L 16.0;
      BLD   102;
      R     "M60.0";
      A     L 16.0;
      BLD   102;
      =     "END_CYCLE";
      A     L 16.0;
      JNB   _021;
      L     0;
      T     "DBWork".PP[1].NumSaldaturaAtt;
_021: NOP   0;
NETWORK
TITLE =
NETWORK
TITLE = delay
      A     "On";
      AN    "FWD_TABLE_ROTATION";
      AN    "REVERSE_TABLE_ROTATION";
      L     S5T#3S;
      SD    "T19";
NETWORK
TITLE = Part on table 1 welding
      A     "On";
      A     "M60.2";
      A     "T19";
      =     L 16.0;
      A     L 16.0;
      A     "DBWork".RotationTable;
      FP    "M1005.7";
      S     "M16.2";
      A     L 16.0;
      AN    "DBWork".RotationTable;
      FP    "M1006.0";
      S     "M16.3";
NETWORK
TITLE = Part on Table 2 Welding
      A     "On";
      A(;
      A     "START_PULSE";
      A     "M26.6";
      O     "M16.1";
      );
      =     L 16.0;
      A     L 16.0;
      A     "DBWork".RotationTable;
      A     "M16.3";
      R     "M16.3";
      A     L 16.0;
      AN    "DBWork".RotationTable;
      A     "M16.2";
      R     "M16.2";
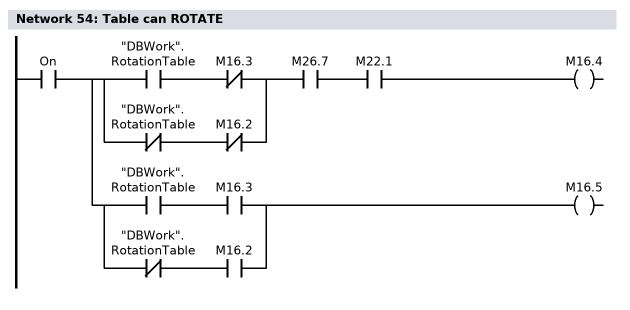
NETWORK
TITLE = Table can ROTATE
      A     "On";
      =     L 16.0;
      A     L 16.0;
      A(;
      A     "DBWork".RotationTable;
      AN    "M16.3";
      O;
      AN    "DBWork".RotationTable;
      AN    "M16.2";
      );
      A     "M26.7";
      A     "M22.1";
      =     "M16.4";
      A     L 16.0;
      A(;
      A     "DBWork".RotationTable;
      A     "M16.3";
      O;
      AN    "DBWork".RotationTable;
      A     "M16.2";
      );
      =     "M16.5";
END_FUNCTION

FUNCTION "FC16 - ALARMS" : VOID	// FC 16
TITLE = Alarms management
VERSION : 0.1
VAR_TEMP
  tempBOOL : BOOL ;
END_VAR
BEGIN
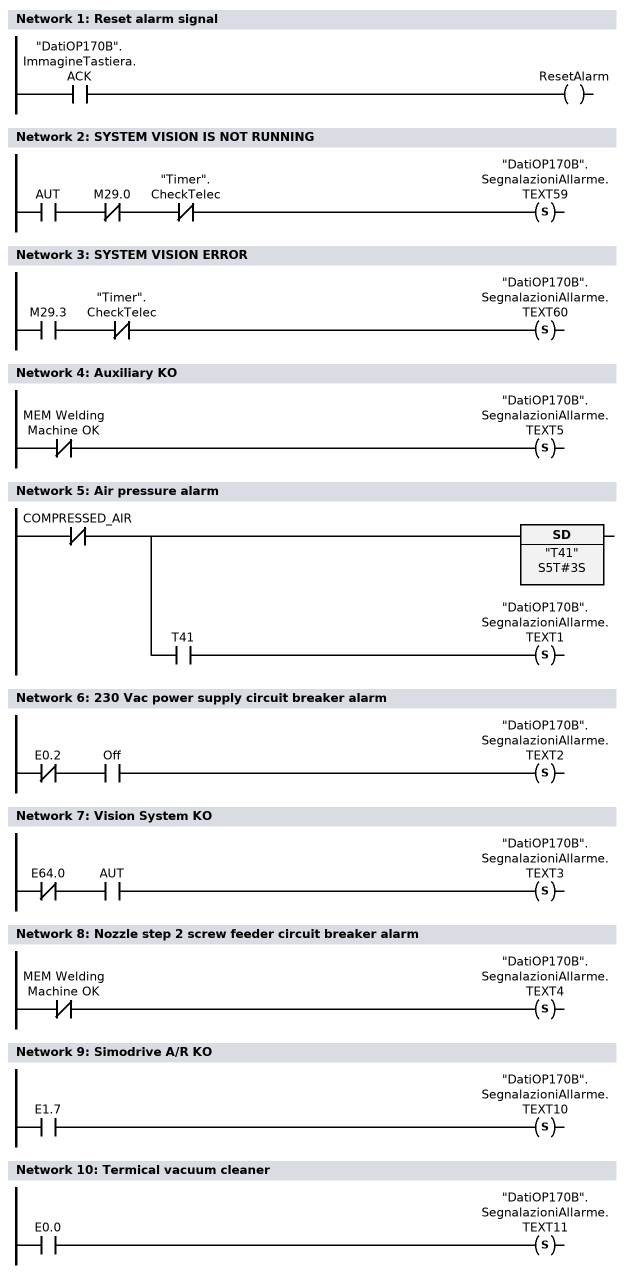
NETWORK
TITLE = Reset alarm signal
      A     "DatiOP170B".ImmagineTastiera.ACK;
      =     "ResetAlarm";
NETWORK
TITLE = SYSTEM VISION IS NOT RUNNING
      A     "AUT";
      AN    "M29.0";
      AN    "Timer".CheckTelec;
      S     "DatiOP170B".SegnalazioniAllarme.TEXT59;
NETWORK
TITLE = SYSTEM VISION ERROR
      A     "M29.3";
      AN    "Timer".CheckTelec;
      S     "DatiOP170B".SegnalazioniAllarme.TEXT60;
NETWORK
TITLE = Auxiliary KO
      AN    "MEM Welding Machine OK";
      S     "DatiOP170B".SegnalazioniAllarme.TEXT5;
NETWORK
TITLE = Air pressure alarm
      AN    "COMPRESSED_AIR";
      =     L 1.0;
      A     L 1.0;
      BLD   102;
      L     S5T#3S;
      SD    "T41";
      A     L 1.0;
      A     "T41";
      S     "DatiOP170B".SegnalazioniAllarme.TEXT1;
NETWORK
TITLE = 230 Vac power supply circuit breaker alarm
      AN    "E0.2";
      A     "Off";
      S     "DatiOP170B".SegnalazioniAllarme.TEXT2;
NETWORK
TITLE = Vision System KO
      AN    "E64.0";
      A     "AUT";
      S     "DatiOP170B".SegnalazioniAllarme.TEXT3;
NETWORK
TITLE = Nozzle step 2 screw feeder circuit breaker alarm
      AN    "MEM Welding Machine OK";
      S     "DatiOP170B".SegnalazioniAllarme.TEXT4;
NETWORK
TITLE = Simodrive A/R KO
      A     "E1.7";
      S     "DatiOP170B".SegnalazioniAllarme.TEXT10;
NETWORK
TITLE = Termical vacuum cleaner
      A     "E0.0";
      S     "DatiOP170B".SegnalazioniAllarme.TEXT11;
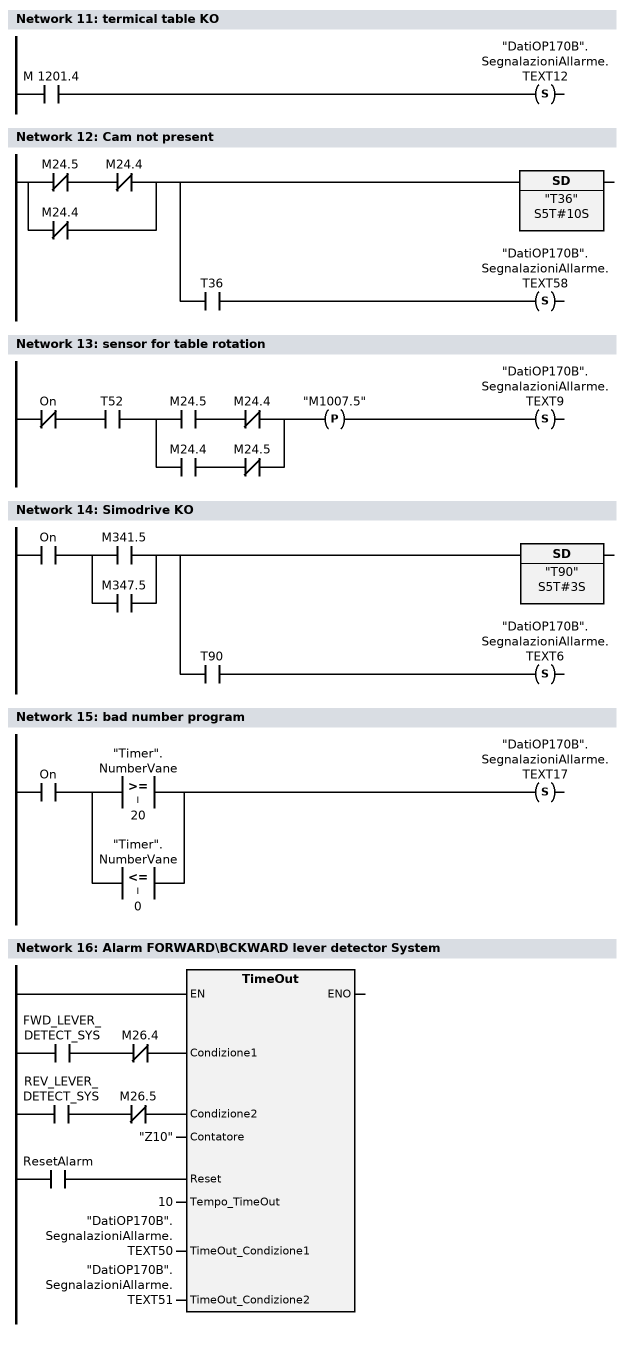
NETWORK
TITLE = termical table KO
      A     M 1201.4;
      S     "DatiOP170B".SegnalazioniAllarme.TEXT12;
NETWORK
TITLE = Cam not present
      AN    "M24.5";
      AN    "M24.4";
      ON    "M24.4";
      =     L 1.0;
      A     L 1.0;
      BLD   102;
      L     S5T#10S;
      SD    "T36";
      A     L 1.0;
      A     "T36";
      S     "DatiOP170B".SegnalazioniAllarme.TEXT58;
NETWORK
TITLE = sensor for table rotation
      AN    "On";
      A     "T52";
      A(;
      A     "M24.5";
      AN    "M24.4";
      O;
      A     "M24.4";
      AN    "M24.5";
      );
      FP    "M1007.5";
      S     "DatiOP170B".SegnalazioniAllarme.TEXT9;
NETWORK
TITLE = Simodrive KO
//press ack button
      A     "On";
      A(;
      O     "M341.5";
      O     "M347.5";
      );
      =     L 1.0;
      A     L 1.0;
      BLD   102;
      L     S5T#3S;
      SD    "T90";
      A     L 1.0;
      A     "T90";
      S     "DatiOP170B".SegnalazioniAllarme.TEXT6;
NETWORK
TITLE = bad number program
      A     "On";
      A(;
      O(;
      L     "Timer".NumberVane;
      L     20;
      >=I;
      );
      O(;
      L     "Timer".NumberVane;
      L     0;
      <=I;
      );
      );
      S     "DatiOP170B".SegnalazioniAllarme.TEXT17;
NETWORK
TITLE = Alarm FORWARD\BCKWARD lever detector System
      A     "FWD_LEVER_DETECT_SYS";
      AN    "M26.4";
      =     L 1.0;
      BLD   103;
      A     "REV_LEVER_DETECT_SYS";
      AN    "M26.5";
      =     L 1.1;
      BLD   103;
      A     "ResetAlarm";
      =     L 1.2;
      BLD   103;
      CALL  "TimeOut" (
           Condizione1              := L 1.0,
           Condizione2              := L 1.1,
           Contatore                := "Z10",
           Reset                    := L 1.2,
           Tempo_TimeOut            := 10,
           TimeOut_Condizione1      := "DatiOP170B".SegnalazioniAllarme.TEXT50,
           TimeOut_Condizione2      := "DatiOP170B".SegnalazioniAllarme.TEXT51);
      NOP   0;
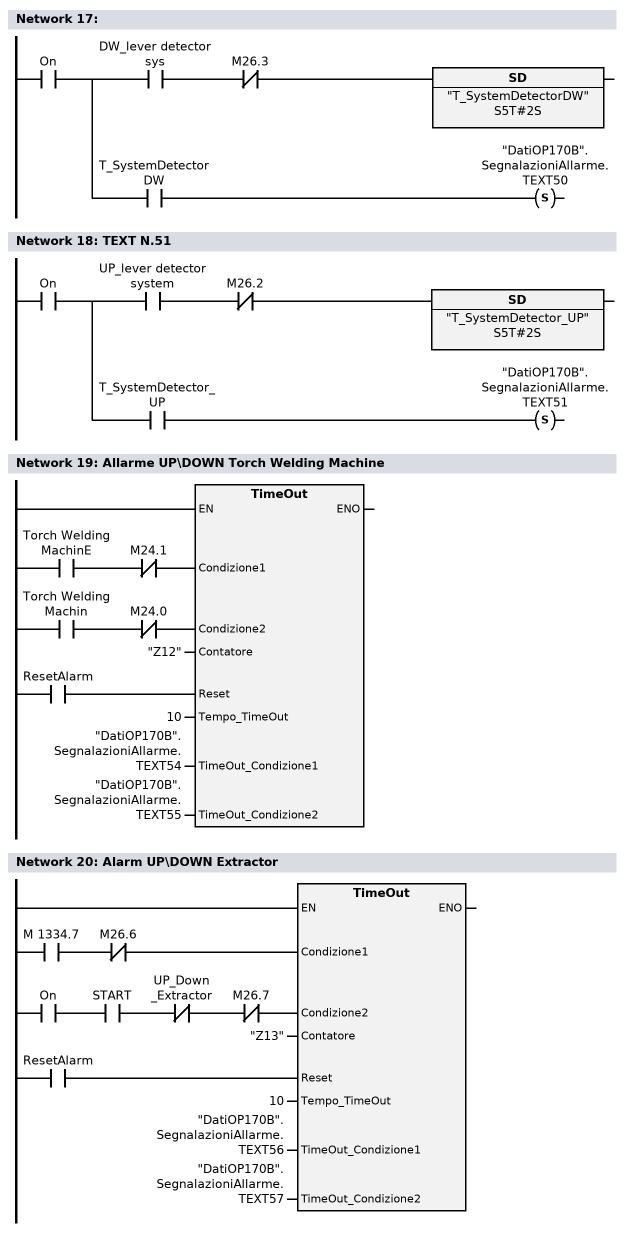
NETWORK
TITLE =
      A     "On";
      =     L 1.0;
      A     L 1.0;
      A     "DW_lever detector sys";
      AN    "M26.3";
      L     S5T#2S;
      SD    "T_SystemDetectorDW";
      A     L 1.0;
      A     "T_SystemDetectorDW";
      S     "DatiOP170B".SegnalazioniAllarme.TEXT50;
NETWORK
TITLE = TEXT N.51
      A     "On";
      =     L 1.0;
      A     L 1.0;
      A     "UP_lever detector system";
      AN    "M26.2";
      L     S5T#2S;
      SD    "T_SystemDetector_UP";
      A     L 1.0;
      A     "T_SystemDetector_UP";
      S     "DatiOP170B".SegnalazioniAllarme.TEXT51;
NETWORK
TITLE = Allarme UP\DOWN Torch Welding Machine
      A     "Torch Welding MachinE";
      AN    "M24.1";
      =     L 1.0;
      BLD   103;
      A     "Torch Welding Machin";
      AN    "M24.0";
      =     L 1.1;
      BLD   103;
      A     "ResetAlarm";
      =     L 1.2;
      BLD   103;
      CALL  "TimeOut" (
           Condizione1              := L 1.0,
           Condizione2              := L 1.1,
           Contatore                := "Z12",
           Reset                    := L 1.2,
           Tempo_TimeOut            := 10,
           TimeOut_Condizione1      := "DatiOP170B".SegnalazioniAllarme.TEXT54,
           TimeOut_Condizione2      := "DatiOP170B".SegnalazioniAllarme.TEXT55);
      NOP   0;
NETWORK
TITLE = Alarm UP\DOWN Extractor
      A     M 1334.7;
      AN    "M26.6";
      =     L 1.0;
      BLD   103;
      A     "On";
      A     "START";
      AN    "UP_Down _Extractor";
      AN    "M26.7";
      =     L 1.1;
      BLD   103;
      A     "ResetAlarm";
      =     L 1.2;
      BLD   103;
      CALL  "TimeOut" (
           Condizione1              := L 1.0,
           Condizione2              := L 1.1,
           Contatore                := "Z13",
           Reset                    := L 1.2,
           Tempo_TimeOut            := 10,
           TimeOut_Condizione1      := "DatiOP170B".SegnalazioniAllarme.TEXT56,
           TimeOut_Condizione2      := "DatiOP170B".SegnalazioniAllarme.TEXT57);
      NOP   0;
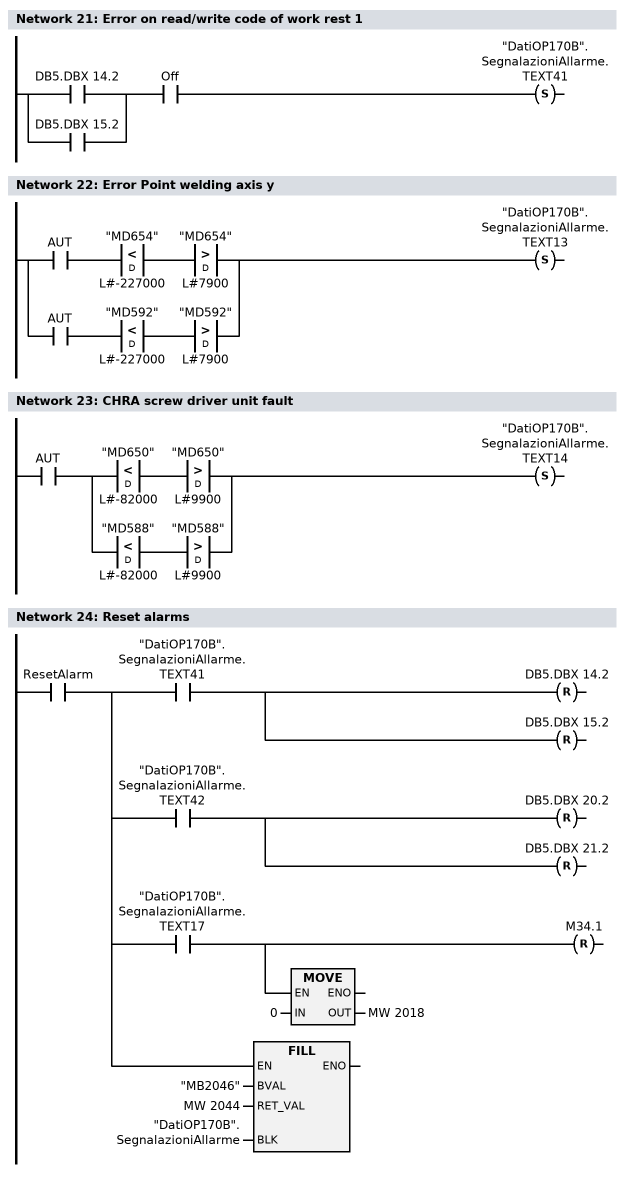
NETWORK
TITLE = Error on read/write code of work rest 1
      A(;
      O     DB5.DBX 14.2;
      O     DB5.DBX 15.2;
      );
      A     "Off";
      S     "DatiOP170B".SegnalazioniAllarme.TEXT41;
NETWORK
TITLE = Error Point welding axis y
      A     "AUT";
      A(;
      L     "MD654";
      L     L#-227000;
      <D;
      );
      A(;
      L     "MD654";
      L     L#7900;
      >D;
      );
      O;
      A     "AUT";
      A(;
      L     "MD592";
      L     L#-227000;
      <D;
      );
      A(;
      L     "MD592";
      L     L#7900;
      >D;
      );
      S     "DatiOP170B".SegnalazioniAllarme.TEXT13;
NETWORK
TITLE = CHRA screw driver unit fault
      A     "AUT";
      A(;
      A(;
      L     "MD650";
      L     L#-82000;
      <D;
      );
      A(;
      L     "MD650";
      L     L#9900;
      >D;
      );
      O;
      A(;
      L     "MD588";
      L     L#-82000;
      <D;
      );
      A(;
      L     "MD588";
      L     L#9900;
      >D;
      );
      );
      S     "DatiOP170B".SegnalazioniAllarme.TEXT14;
NETWORK
TITLE = Reset alarms
      A     "ResetAlarm";
      =     L 1.0;
      A     L 1.0;
      A     "DatiOP170B".SegnalazioniAllarme.TEXT41;
      R     DB5.DBX 14.2;
      R     DB5.DBX 15.2;
      A     L 1.0;
      A     "DatiOP170B".SegnalazioniAllarme.TEXT42;
      R     DB5.DBX 20.2;
      R     DB5.DBX 21.2;
      A     L 1.0;
      A     "DatiOP170B".SegnalazioniAllarme.TEXT17;
      =     L 1.1;
      A     L 1.1;
      BLD   102;
      R     "M34.1";
      A     L 1.1;
      JNB   _001;
      L     0;
      T     MW 2018;
_001: NOP   0;
      A     L 1.0;
      JNB   _002;
      CALL  "FILL" (
           BVAL                     := "MB2046",
           RET_VAL                  := MW 2044,
           BLK                      := "DatiOP170B".SegnalazioniAllarme);
_002: NOP   0;
NETWORK
TITLE = Spacer circular feeder empty
      CLR;
      =     "DatiOP170B".SegnalazioniAllarme.TEXT15;
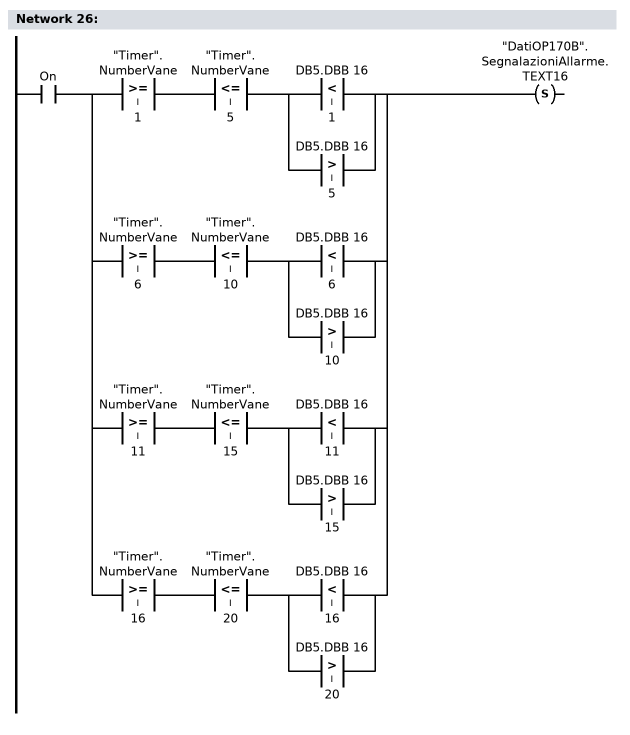
NETWORK
TITLE =
      A     "On";
      A(;
      A(;
      L     "Timer".NumberVane;
      L     1;
      >=I;
      );
      A(;
      L     "Timer".NumberVane;
      L     5;
      <=I;
      );
      A(;
      O(;
      L     DB5.DBB 16;
      L     1;
      <I;
      );
      O(;
      L     DB5.DBB 16;
      L     5;
      >I;
      );
      );
      O;
      A(;
      L     "Timer".NumberVane;
      L     6;
      >=I;
      );
      A(;
      L     "Timer".NumberVane;
      L     10;
      <=I;
      );
      A(;
      O(;
      L     DB5.DBB 16;
      L     6;
      <I;
      );
      O(;
      L     DB5.DBB 16;
      L     10;
      >I;
      );
      );
      O;
      A(;
      L     "Timer".NumberVane;
      L     11;
      >=I;
      );
      A(;
      L     "Timer".NumberVane;
      L     15;
      <=I;
      );
      A(;
      O(;
      L     DB5.DBB 16;
      L     11;
      <I;
      );
      O(;
      L     DB5.DBB 16;
      L     15;
      >I;
      );
      );
      O;
      A(;
      L     "Timer".NumberVane;
      L     16;
      >=I;
      );
      A(;
      L     "Timer".NumberVane;
      L     20;
      <=I;
      );
      A(;
      O(;
      L     DB5.DBB 16;
      L     16;
      <I;
      );
      O(;
      L     DB5.DBB 16;
      L     20;
      >I;
      );
      );
      );
      S     "DatiOP170B".SegnalazioniAllarme.TEXT16;
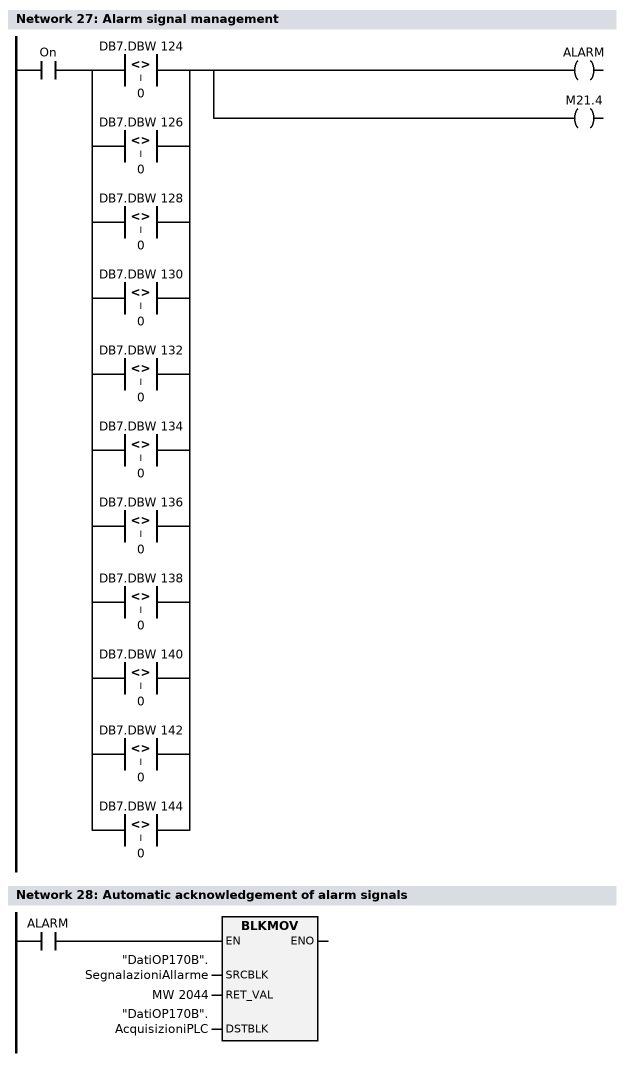
NETWORK
TITLE = Alarm signal management
      A     "On";
      A(;
      O(;
      L     DB7.DBW 124;
      L     0;
      <>I;
      );
      O(;
      L     DB7.DBW 126;
      L     0;
      <>I;
      );
      O(;
      L     DB7.DBW 128;
      L     0;
      <>I;
      );
      O(;
      L     DB7.DBW 130;
      L     0;
      <>I;
      );
      O(;
      L     DB7.DBW 132;
      L     0;
      <>I;
      );
      O(;
      L     DB7.DBW 134;
      L     0;
      <>I;
      );
      O(;
      L     DB7.DBW 136;
      L     0;
      <>I;
      );
      O(;
      L     DB7.DBW 138;
      L     0;
      <>I;
      );
      O(;
      L     DB7.DBW 140;
      L     0;
      <>I;
      );
      O(;
      L     DB7.DBW 142;
      L     0;
      <>I;
      );
      O(;
      L     DB7.DBW 144;
      L     0;
      <>I;
      );
      );
      =     "ALARM";
      =     "M21.4";
NETWORK
TITLE = Automatic acknowledgement of alarm signals
      A     "ALARM";
      JNB   _003;
      CALL  "BLKMOV" (
           SRCBLK                   := "DatiOP170B".SegnalazioniAllarme,
           RET_VAL                  := MW 2044,
           DSTBLK                   := "DatiOP170B".AcquisizioniPLC);
_003: NOP   0;
END_FUNCTION

FUNCTION "FC17 - OPERATOR PANNEL" : VOID	// FC 17
TITLE = OP170B Operator Pannel Interface
VERSION : 0.1
BEGIN
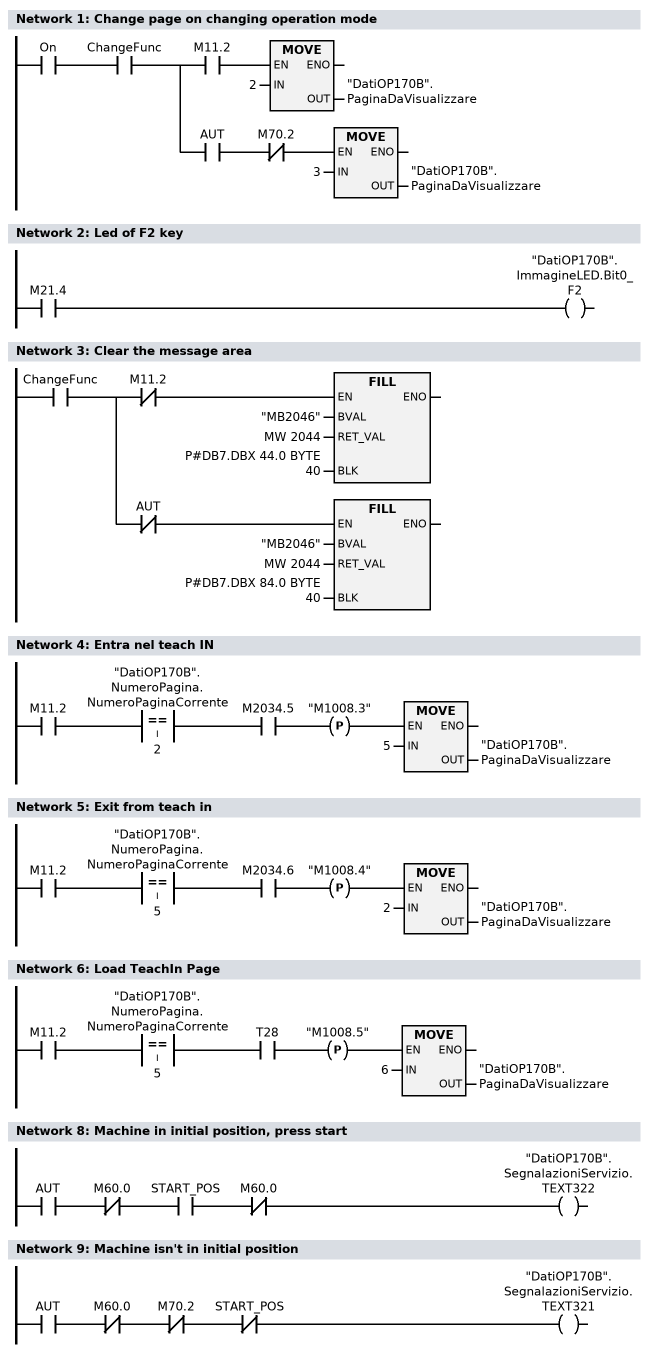
NETWORK
TITLE = Change page on changing operation mode
      A     "On";
      A     "ChangeFunc";
      =     L 0.0;
      A     L 0.0;
      A     "M11.2";
      JNB   _001;
      L     2;
      T     "DatiOP170B".PaginaDaVisualizzare;
_001: NOP   0;
      A     L 0.0;
      A     "AUT";
      AN    "M70.2";
      JNB   _002;
      L     3;
      T     "DatiOP170B".PaginaDaVisualizzare;
_002: NOP   0;
NETWORK
TITLE = Led of F2 key
      A     "M21.4";
      =     "DatiOP170B".ImmagineLED.Bit0_F2;
NETWORK
TITLE = Clear the message area
      A     "ChangeFunc";
      =     L 0.0;
      A     L 0.0;
      AN    "M11.2";
      JNB   _003;
      CALL  "FILL" (
           BVAL                     := "MB2046",
           RET_VAL                  := MW 2044,
           BLK                      := P#DB7.DBX 44.0 BYTE 40);
_003: NOP   0;
      A     L 0.0;
      AN    "AUT";
      JNB   _004;
      CALL  "FILL" (
           BVAL                     := "MB2046",
           RET_VAL                  := MW 2044,
           BLK                      := P#DB7.DBX 84.0 BYTE 40);
_004: NOP   0;
NETWORK
TITLE = Entra nel teach IN
      A     "M11.2";
      A(;
      L     "DatiOP170B".NumeroPagina.NumeroPaginaCorrente;
      L     2;
      ==I;
      );
      A     "M2034.5";
      FP    "M1008.3";
      JNB   _005;
      L     5;
      T     "DatiOP170B".PaginaDaVisualizzare;
_005: NOP   0;
NETWORK
TITLE = Exit from teach in
      A     "M11.2";
      A(;
      L     "DatiOP170B".NumeroPagina.NumeroPaginaCorrente;
      L     5;
      ==I;
      );
      A     "M2034.6";
      FP    "M1008.4";
      JNB   _006;
      L     2;
      T     "DatiOP170B".PaginaDaVisualizzare;
_006: NOP   0;
NETWORK
TITLE = Load TeachIn Page
//Aspetto il T28 in modo tale da lanciare il comando agli assi
      A     "M11.2";
      A(;
      L     "DatiOP170B".NumeroPagina.NumeroPaginaCorrente;
      L     5;
      ==I;
      );
      A     "T28";
      FP    "M1008.5";
      JNB   _007;
      L     6;
      T     "DatiOP170B".PaginaDaVisualizzare;
_007: NOP   0;
NETWORK
TITLE =
NETWORK
TITLE = Machine in initial position, press start
      A     "AUT";
      AN    "M60.0";
      A     "START_POS";
      AN    "M60.0";
      =     "DatiOP170B".SegnalazioniServizio.TEXT322;
NETWORK
TITLE = Machine isn't in initial position
      A     "AUT";
      AN    "M60.0";
      AN    "M70.2";
      AN    "START_POS";
      =     "DatiOP170B".SegnalazioniServizio.TEXT321;
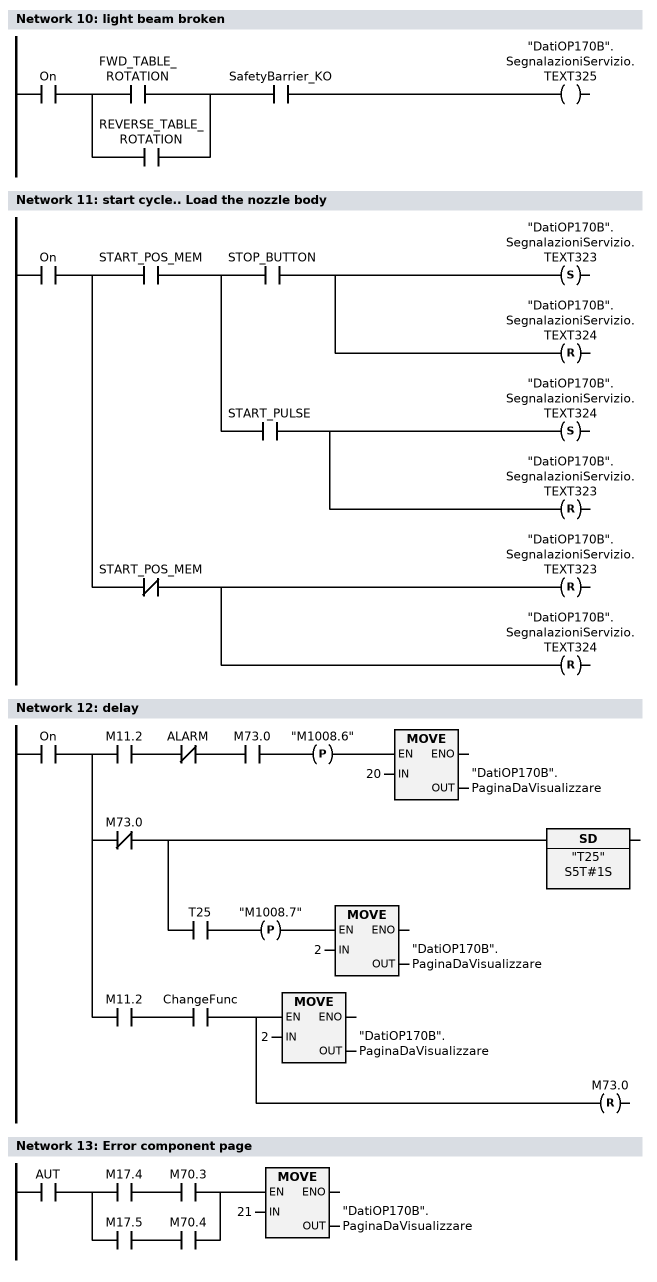
NETWORK
TITLE = light beam broken
      A     "On";
      A(;
      O     "FWD_TABLE_ROTATION";
      O     "REVERSE_TABLE_ROTATION";
      );
      A     "SafetyBarrier_KO";
      =     "DatiOP170B".SegnalazioniServizio.TEXT325;
NETWORK
TITLE = start cycle.. Load the nozzle body
      A     "On";
      =     L 0.0;
      A     L 0.0;
      A     "START_POS_MEM";
      =     L 0.1;
      A     L 0.1;
      A     "STOP_BUTTON";
      S     "DatiOP170B".SegnalazioniServizio.TEXT323;
      R     "DatiOP170B".SegnalazioniServizio.TEXT324;
      A     L 0.1;
      A     "START_PULSE";
      S     "DatiOP170B".SegnalazioniServizio.TEXT324;
      R     "DatiOP170B".SegnalazioniServizio.TEXT323;
      A     L 0.0;
      AN    "START_POS_MEM";
      R     "DatiOP170B".SegnalazioniServizio.TEXT323;
      R     "DatiOP170B".SegnalazioniServizio.TEXT324;
NETWORK
TITLE = delay
//Page of repositioning
      A     "On";
      =     L 0.0;
      A     L 0.0;
      A     "M11.2";
      AN    "ALARM";
      A     "M73.0";
      FP    "M1008.6";
      JNB   _008;
      L     20;
      T     "DatiOP170B".PaginaDaVisualizzare;
_008: NOP   0;
      A     L 0.0;
      AN    "M73.0";
      =     L 0.1;
      A     L 0.1;
      BLD   102;
      L     S5T#1S;
      SD    "T25";
      A     L 0.1;
      A     "T25";
      FP    "M1008.7";
      JNB   _009;
      L     2;
      T     "DatiOP170B".PaginaDaVisualizzare;
_009: NOP   0;
      A     L 0.0;
      A     "M11.2";
      A     "ChangeFunc";
      =     L 0.1;
      A     L 0.1;
      JNB   _00a;
      L     2;
      T     "DatiOP170B".PaginaDaVisualizzare;
_00a: NOP   0;
      A     L 0.1;
      BLD   102;
      R     "M73.0";
NETWORK
TITLE = Error component page
      A     "AUT";
      A(;
      A     "M17.4";
      A     "M70.3";
      O;
      A     "M17.5";
      A     "M70.4";
      );
      JNB   _00b;
      L     21;
      T     "DatiOP170B".PaginaDaVisualizzare;
_00b: NOP   0;
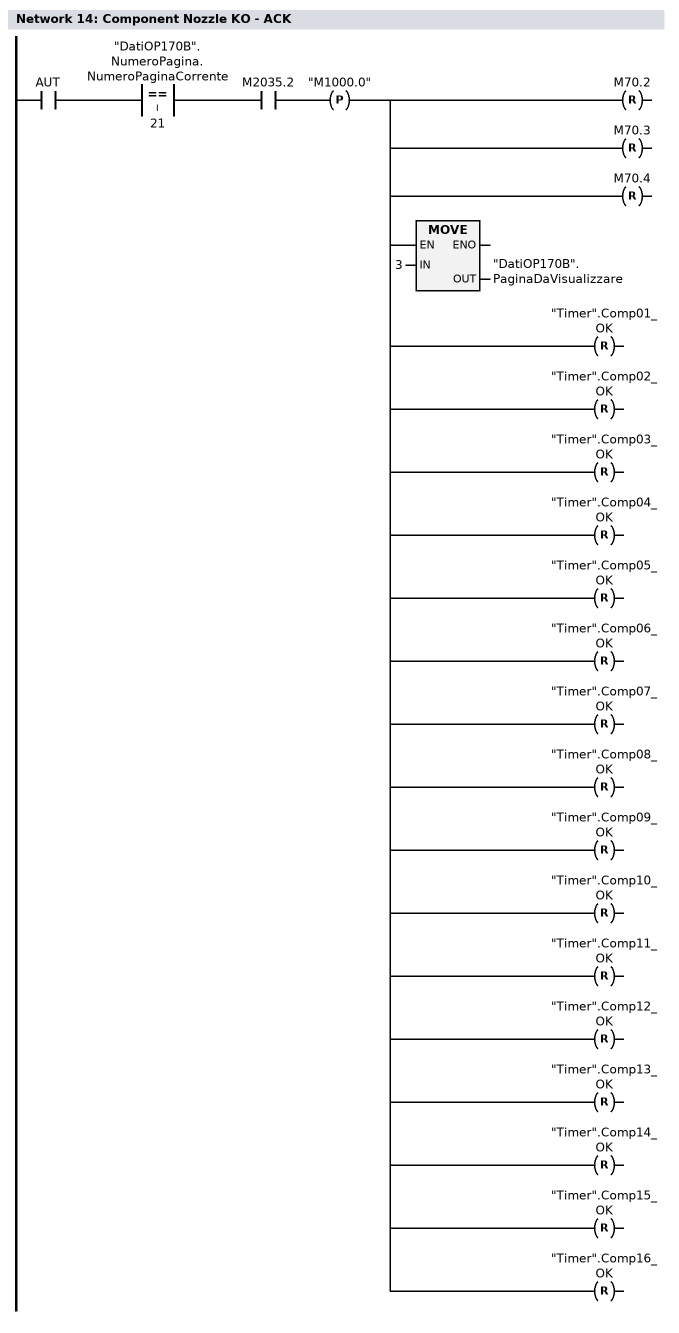
NETWORK
TITLE = Component Nozzle KO - ACK
      A     "AUT";
      A(;
      L     "DatiOP170B".NumeroPagina.NumeroPaginaCorrente;
      L     21;
      ==I;
      );
      A     "M2035.2";
      FP    "M1000.0";
      =     L 0.0;
      A     L 0.0;
      BLD   102;
      R     "M70.2";
      A     L 0.0;
      BLD   102;
      R     "M70.3";
      A     L 0.0;
      BLD   102;
      R     "M70.4";
      A     L 0.0;
      JNB   _00c;
      L     3;
      T     "DatiOP170B".PaginaDaVisualizzare;
_00c: NOP   0;
      A     L 0.0;
      BLD   102;
      R     "Timer".Comp01_OK;
      A     L 0.0;
      BLD   102;
      R     "Timer".Comp02_OK;
      A     L 0.0;
      BLD   102;
      R     "Timer".Comp03_OK;
      A     L 0.0;
      BLD   102;
      R     "Timer".Comp04_OK;
      A     L 0.0;
      BLD   102;
      R     "Timer".Comp05_OK;
      A     L 0.0;
      BLD   102;
      R     "Timer".Comp06_OK;
      A     L 0.0;
      BLD   102;
      R     "Timer".Comp07_OK;
      A     L 0.0;
      BLD   102;
      R     "Timer".Comp08_OK;
      A     L 0.0;
      BLD   102;
      R     "Timer".Comp09_OK;
      A     L 0.0;
      BLD   102;
      R     "Timer".Comp10_OK;
      A     L 0.0;
      BLD   102;
      R     "Timer".Comp11_OK;
      A     L 0.0;
      BLD   102;
      R     "Timer".Comp12_OK;
      A     L 0.0;
      BLD   102;
      R     "Timer".Comp13_OK;
      A     L 0.0;
      BLD   102;
      R     "Timer".Comp14_OK;
      A     L 0.0;
      BLD   102;
      R     "Timer".Comp15_OK;
      A     L 0.0;
      BLD   102;
      R     "Timer".Comp16_OK;
